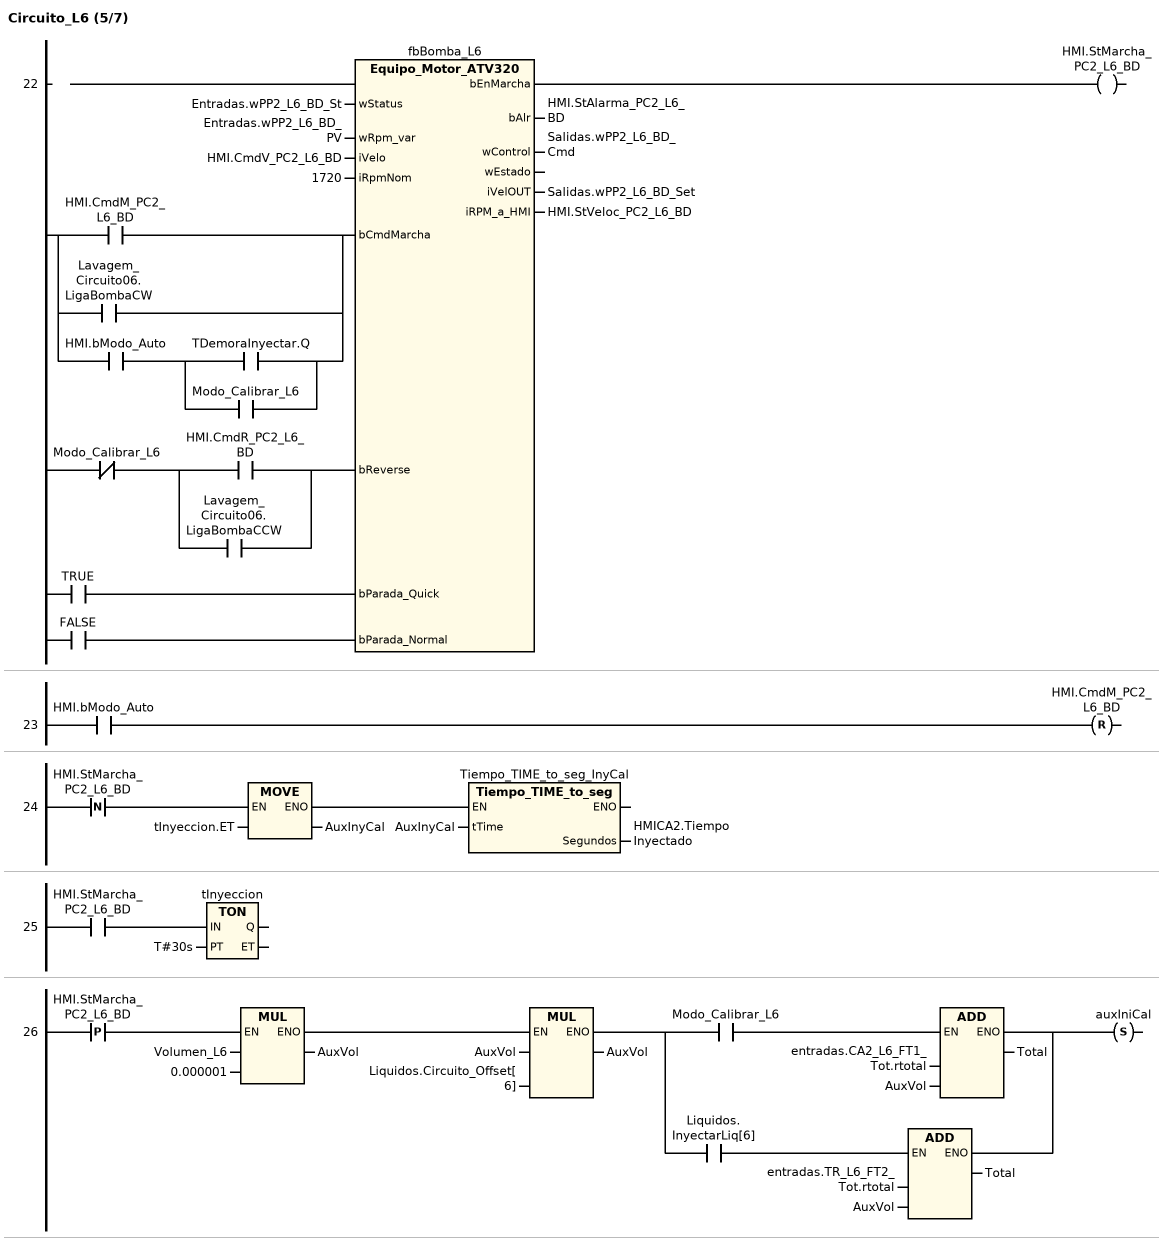
// NETWORK 22
fbBomba_L6(
    wStatus := Entradas.wPP2_L6_BD_St,
    wRpm_var := Entradas.wPP2_L6_BD_PV,
    iVelo := HMI.CmdV_PC2_L6_BD,
    iRpmNom := 1720,
    bCmdMarcha := HMI.CmdM_PC2_L6_BD OR Lavagem_Circuito06.LigaBombaCW OR HMI.bModo_Auto AND (TDemoraInyectar.Q OR Modo_Calibrar_L6),
    bReverse := NOT Modo_Calibrar_L6 AND (HMI.CmdR_PC2_L6_BD OR Lavagem_Circuito06.LigaBombaCCW),
    bParada_Quick := TRUE,
    bParada_Normal := FALSE,
    bAlr => HMI.StAlarma_PC2_L6_BD,
    wControl => Salidas.wPP2_L6_BD_Cmd,
    iVelOUT => Salidas.wPP2_L6_BD_Set,
    iRPM_a_HMI => HMI.StVeloc_PC2_L6_BD); // Equipo_Motor_ATV320
HMI.StMarcha_PC2_L6_BD := fbBomba_L6.bEnMarcha;

// NETWORK 23
HMI.CmdM_PC2_L6_BD R= HMI.bModo_Auto;

// NETWORK 24
_ft1(CLK := HMI.StMarcha_PC2_L6_BD);
_w8 := _ft1.Q;
IF _w8 THEN AuxInyCal := tInyeccion.ET; END_IF
IF _w8 THEN
    Tiempo_TIME_to_seg_InyCal(tTime := AuxInyCal, Segundos => HMICA2.TiempoInyectado); // Tiempo_TIME_to_seg
END_IF

// NETWORK 25
tInyeccion(IN := HMI.StMarcha_PC2_L6_BD, PT := T#30s); // TON

// NETWORK 26
_rt1(CLK := HMI.StMarcha_PC2_L6_BD);
_w9 := _rt1.Q;
IF _w9 THEN AuxVol := Volumen_L6 * 0.000001; END_IF
IF _w9 THEN AuxVol := AuxVol * Liquidos.Circuito_Offset[6]; END_IF
IF _w9 AND Modo_Calibrar_L6 THEN Total := entradas.CA2_L6_FT1_Tot.rtotal + AuxVol; END_IF
IF _w9 AND Liquidos.InyectarLiq[6] THEN Total := entradas.TR_L6_FT2_Tot.rtotal + AuxVol; END_IF
auxIniCal S= _w9 AND Modo_Calibrar_L6 OR _w9 AND Liquidos.InyectarLiq[6];

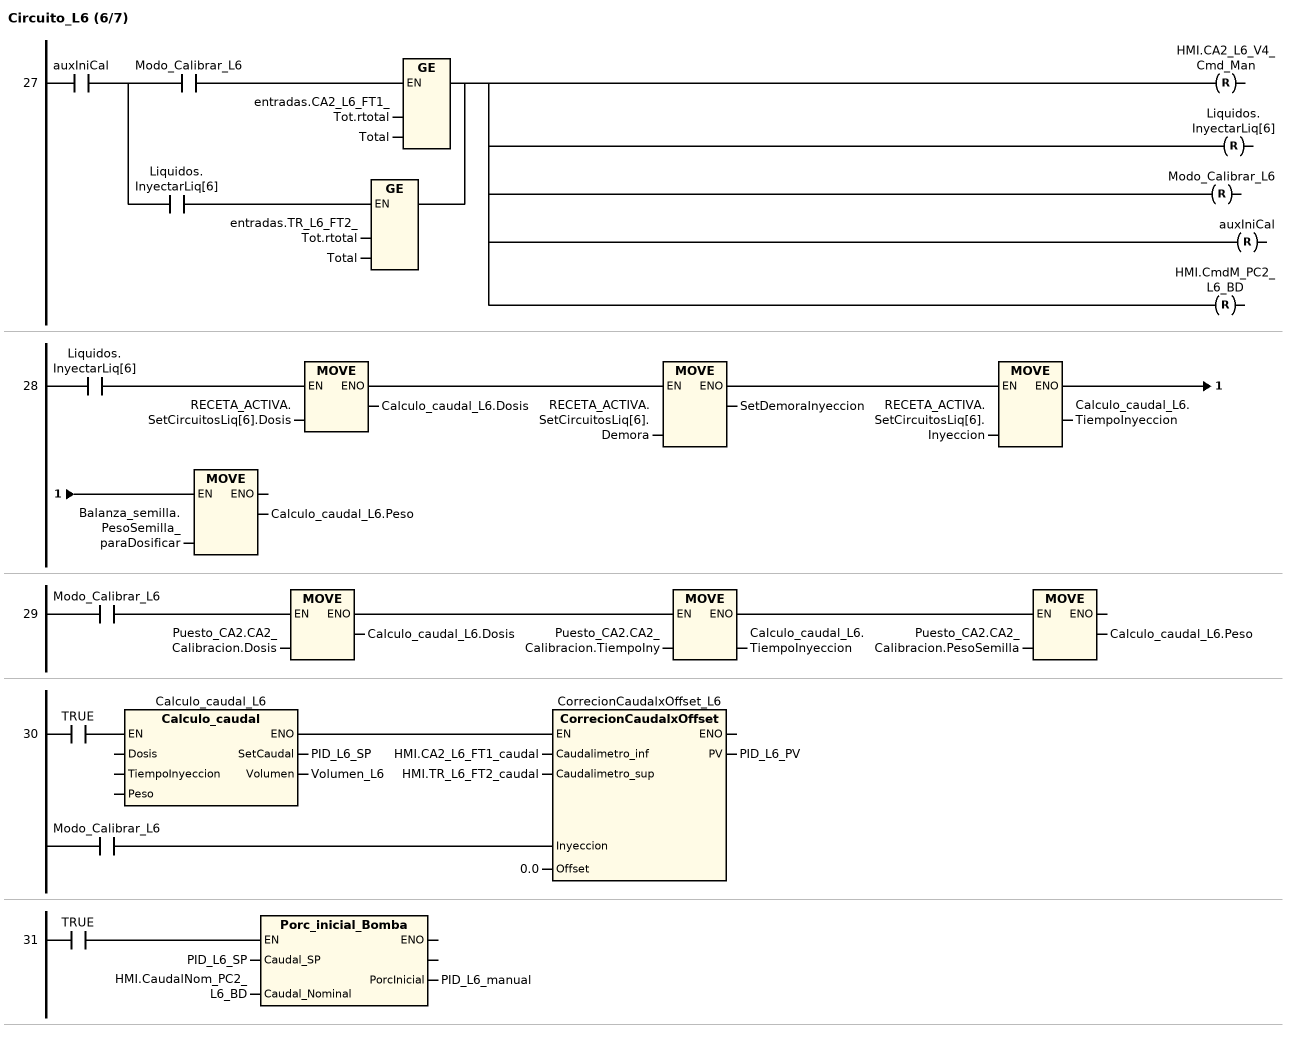
// NETWORK 27
_w10 := auxIniCal AND Modo_Calibrar_L6 AND entradas.CA2_L6_FT1_Tot.rtotal >= Total OR auxIniCal AND Liquidos.InyectarLiq[6] AND entradas.TR_L6_FT2_Tot.rtotal >= Total;
HMI.CA2_L6_V4_Cmd_Man R= _w10;
Liquidos.InyectarLiq[6] R= _w10;
Modo_Calibrar_L6 R= _w10;
auxIniCal R= _w10;
HMI.CmdM_PC2_L6_BD R= _w10;

// NETWORK 28
_w11 := Liquidos.InyectarLiq[6];
IF _w11 THEN Calculo_caudal_L6.Dosis := RECETA_ACTIVA.SetCircuitosLiq[6].Dosis; END_IF
IF _w11 THEN SetDemoraInyeccion := RECETA_ACTIVA.SetCircuitosLiq[6].Demora; END_IF
IF _w11 THEN Calculo_caudal_L6.TiempoInyeccion := RECETA_ACTIVA.SetCircuitosLiq[6].Inyeccion; END_IF
IF _w11 THEN Calculo_caudal_L6.Peso := Balanza_semilla.PesoSemilla_paraDosificar; END_IF

// NETWORK 29
_w12 := Modo_Calibrar_L6;
IF _w12 THEN Calculo_caudal_L6.Dosis := Puesto_CA2.CA2_Calibracion.Dosis; END_IF
IF _w12 THEN Calculo_caudal_L6.TiempoInyeccion := Puesto_CA2.CA2_Calibracion.TiempoIny; END_IF
IF _w12 THEN Calculo_caudal_L6.Peso := Puesto_CA2.CA2_Calibracion.PesoSemilla; END_IF

// NETWORK 30
Calculo_caudal_L6(SetCaudal => PID_L6_SP, Volumen => Volumen_L6); // Calculo_caudal
CorrecionCaudalxOffset_L6(
    Caudalimetro_inf := HMI.CA2_L6_FT1_caudal,
    Caudalimetro_sup := HMI.TR_L6_FT2_caudal,
    Inyeccion := Modo_Calibrar_L6,
    Offset := 0.0,
    PV => PID_L6_PV); // CorrecionCaudalxOffset

// NETWORK 31
Porc_inicial_Bomba(Caudal_SP := PID_L6_SP, Caudal_Nominal := HMI.CaudalNom_PC2_L6_BD, PorcInicial => PID_L6_manual);

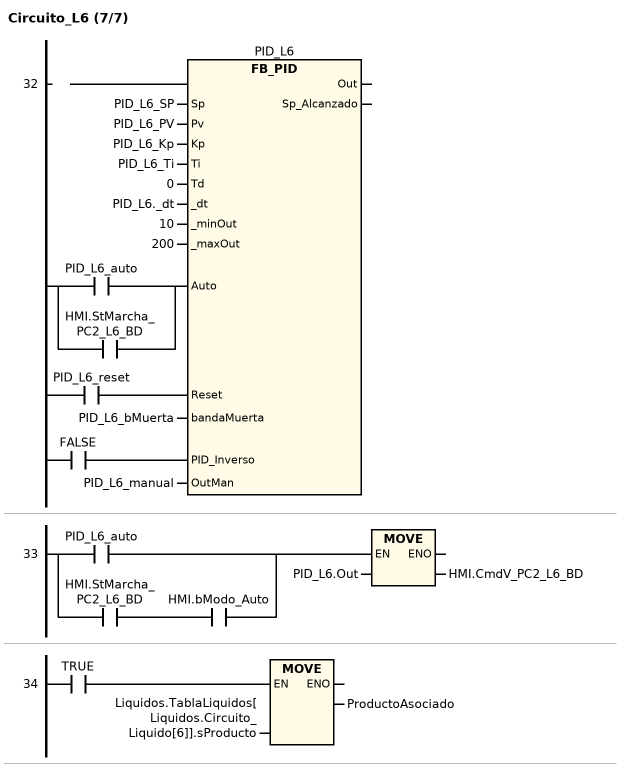
// NETWORK 32
PID_L6(
    Sp := PID_L6_SP,
    Pv := PID_L6_PV,
    Kp := PID_L6_Kp,
    Ti := PID_L6_Ti,
    Td := 0,
    _dt := PID_L6._dt,
    _minOut := 10,
    _maxOut := 200,
    Auto := PID_L6_auto OR HMI.StMarcha_PC2_L6_BD,
    Reset := PID_L6_reset,
    bandaMuerta := PID_L6_bMuerta,
    PID_Inverso := FALSE,
    OutMan := PID_L6_manual); // FB_PID

// NETWORK 33
IF PID_L6_auto OR HMI.StMarcha_PC2_L6_BD AND HMI.bModo_Auto THEN HMI.CmdV_PC2_L6_BD := PID_L6.Out; END_IF

// NETWORK 34
ProductoAsociado := Liquidos.TablaLiquidos[Liquidos.Circuito_Liquido[6]].sProducto;

END_PROGRAM

// ---- POUs/Puesto_Calibracion_2/Circuito_L7.TcPOU
PROGRAM Circuito_L7
VAR_INPUT
	Modo_Calibrar_L7: BOOL;
END_VAR
VAR
		fbBomba_L7 :Equipo_Motor_ATV320;
		ControlValv_ioLink_V1:ControlValv_ioLink;
		ControlValv_ioLink_V2: ControlValv_ioLink;
		ControlValv_ioLink_V3: ControlValv_ioLink;
		ControlValv_ioLink_V4: ControlValv_ioLink;
		Falla_L7_V1:BOOL;
		Falla_L7_V2:BOOL;
		Falla_L7_V3:BOOL;
		Falla_L7_V4:BOOL;
	Balanza_PU2_WT7: Balanza;
		dHS:DINT;
		TOF_calibradoIBC: TOF;
		PID_L7_SP:REAL;
		PID_L7_auto:BOOL;
		PID_L7_reset:BOOL;
		PID_L7_manual:REAL;
		PID_L7_bMuerta:REAL := 5;
		PID_L7_Kp:REAL := 0.1;
		PID_L7_Ti:REAL := 100;
		PID_L7_PV:REAL;
		Dosis_L7	:REAL;
		TiempoInyeccion_L7	:DINT;
		Peso	:REAL;
		Offset_L7:REAL;
		Inyeccion_L7:BOOL;
		Volumen_L7:REAL;
		Calculo_caudal_L7: Calculo_caudal;
		CorrecionCaudalxOffset_L7: CorrecionCaudalxOffset;
		tInyeccion: TON;
		Total :REAL;
		Totalant	:REAL;
		auxIniCal:BOOL;
		AuxVol:REAL;
		CA2_L7_V1_CmdA_Man :BOOL;
		CA2_L7_V4_CmdA_Man :BOOL;
		TDemoraInyectar: TON;
		SetDemoraInyeccion: REAL;
		Tiempo_seg_to_TIME_DemoraInyec: Tiempo_seg_to_TIME;
		AuxTDemoraInyec: TIME;
		PID_L7: FB_PID;
		Tiempo_TIME_to_seg_InyCal: Tiempo_TIME_to_seg;
		AuxInyCal:TIME;		
		IniTotalFT2:REAL;
		Auxconsumo:REAL;	
	ProductoAsociado: STRING;
	Lavagem_Circuito07: Lavagem;
	Calibracao_teste: Calibracao_V03;
END_VAR

VAR PERSISTENT
	UltimaCalibracao	:UDINT;	//Data e hora da ultima calibração
END_VAR
VAR // added by the converter: edge detectors and wires of the graphical bodies
    _w1, _w2, _w3, _w4, _w5, _w6, _w7, _w8, _w9, _w10, _w11, _w12, _w13 : BOOL;
    _ft1 : F_TRIG;
    _rt1, _rt2 : R_TRIG;
END_VAR

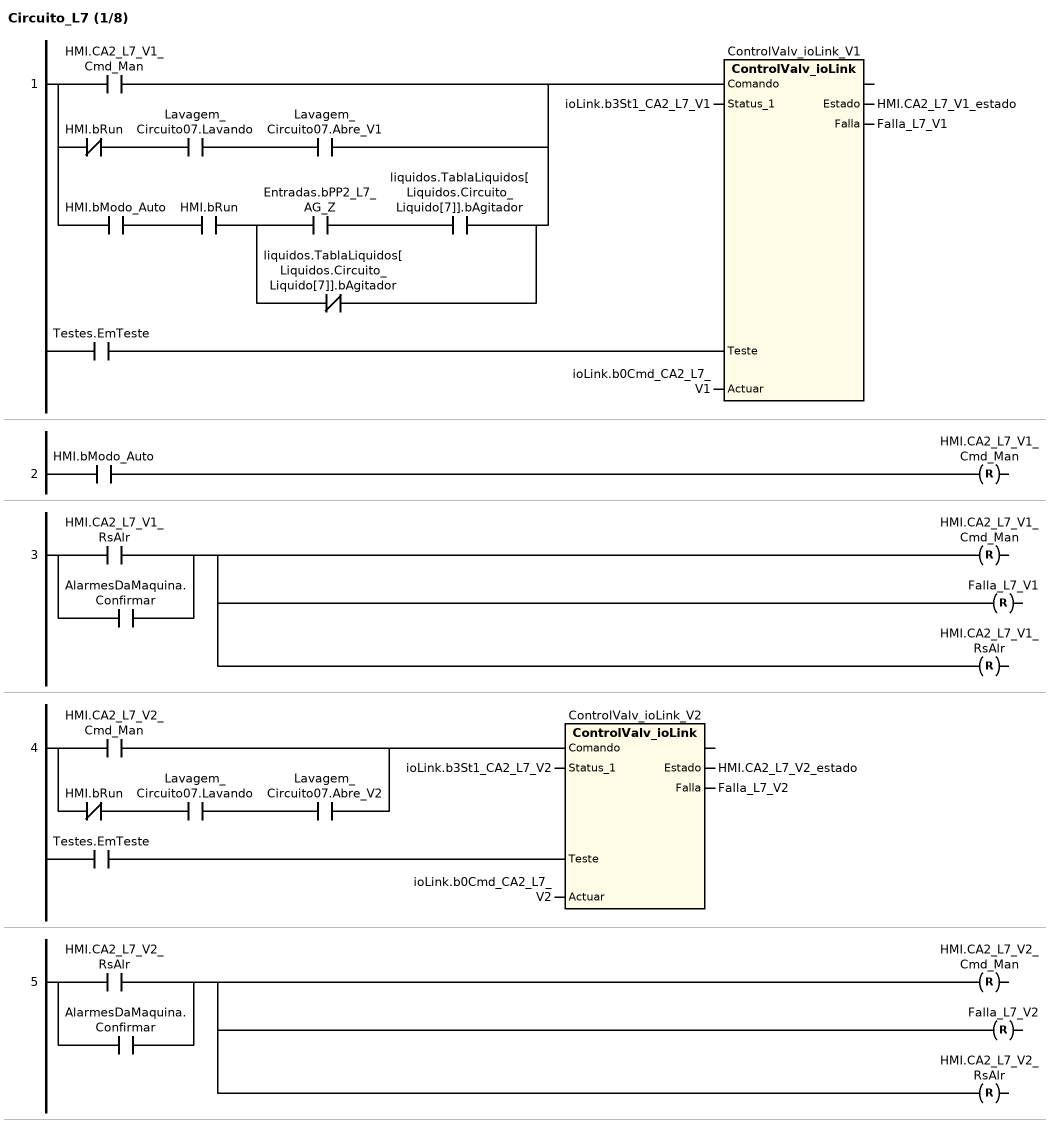
// NETWORK 1
ControlValv_ioLink_V1(
    Comando := HMI.CA2_L7_V1_Cmd_Man OR NOT HMI.bRun AND Lavagem_Circuito07.Lavando AND Lavagem_Circuito07.Abre_V1 OR HMI.bModo_Auto AND HMI.bRun AND (Entradas.bPP2_L7_AG_Z AND (liquidos.TablaLiquidos[Liquidos.Circuito_Liquido[7]].bAgitador) OR NOT (liquidos.TablaLiquidos[Liquidos.Circuito_Liquido[7]].bAgitador)),
    Status_1 := ioLink.b3St1_CA2_L7_V1,
    Teste := Testes.EmTeste,
    Actuar := ioLink.b0Cmd_CA2_L7_V1,
    Estado => HMI.CA2_L7_V1_estado,
    Falla => Falla_L7_V1); // ControlValv_ioLink

// NETWORK 2
HMI.CA2_L7_V1_Cmd_Man R= HMI.bModo_Auto;

// NETWORK 3
_w1 := HMI.CA2_L7_V1_RsAlr OR AlarmesDaMaquina.Confirmar;
HMI.CA2_L7_V1_Cmd_Man R= _w1;
Falla_L7_V1 R= _w1;
HMI.CA2_L7_V1_RsAlr R= _w1;

// NETWORK 4
ControlValv_ioLink_V2(
    Comando := HMI.CA2_L7_V2_Cmd_Man OR NOT HMI.bRun AND Lavagem_Circuito07.Lavando AND Lavagem_Circuito07.Abre_V2,
    Status_1 := ioLink.b3St1_CA2_L7_V2,
    Teste := Testes.EmTeste,
    Actuar := ioLink.b0Cmd_CA2_L7_V2,
    Estado => HMI.CA2_L7_V2_estado,
    Falla => Falla_L7_V2); // ControlValv_ioLink

// NETWORK 5
_w2 := HMI.CA2_L7_V2_RsAlr OR AlarmesDaMaquina.Confirmar;
HMI.CA2_L7_V2_Cmd_Man R= _w2;
Falla_L7_V2 R= _w2;
HMI.CA2_L7_V2_RsAlr R= _w2;

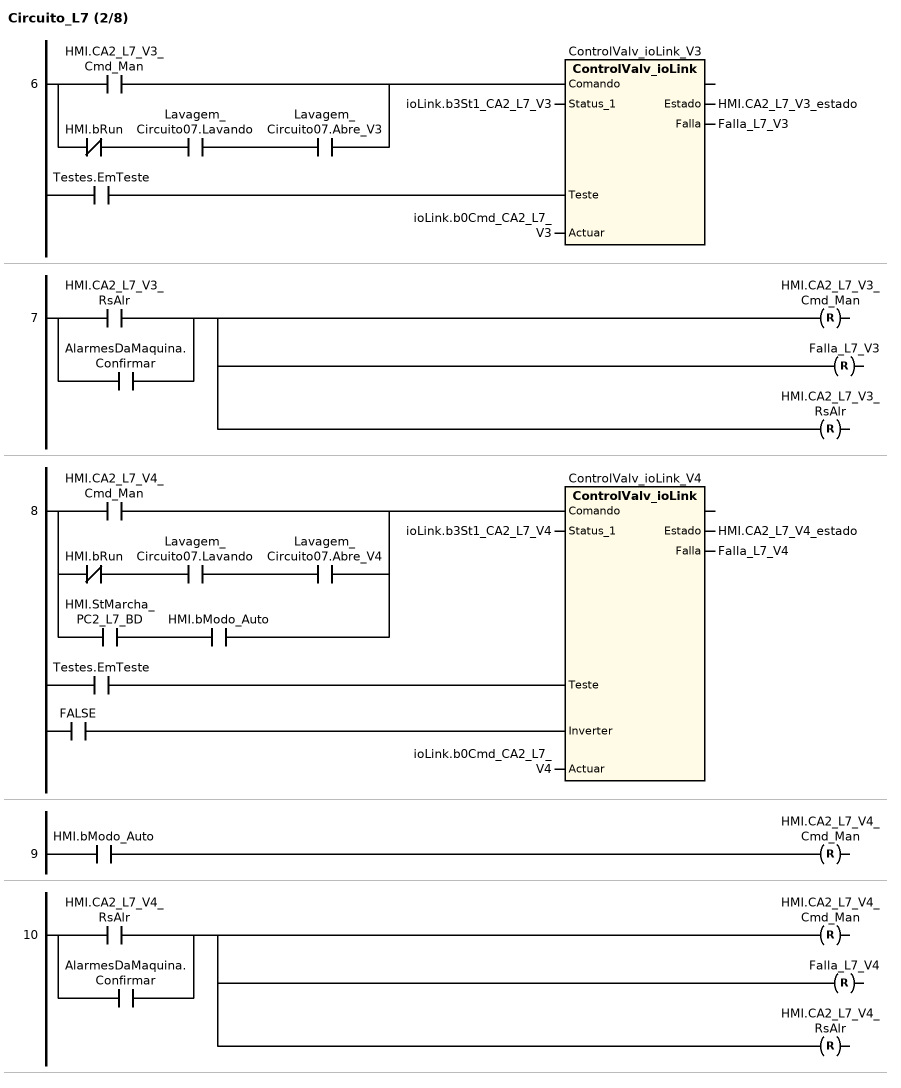
// NETWORK 6
ControlValv_ioLink_V3(
    Comando := HMI.CA2_L7_V3_Cmd_Man OR NOT HMI.bRun AND Lavagem_Circuito07.Lavando AND Lavagem_Circuito07.Abre_V3,
    Status_1 := ioLink.b3St1_CA2_L7_V3,
    Teste := Testes.EmTeste,
    Actuar := ioLink.b0Cmd_CA2_L7_V3,
    Estado => HMI.CA2_L7_V3_estado,
    Falla => Falla_L7_V3); // ControlValv_ioLink

// NETWORK 7
_w3 := HMI.CA2_L7_V3_RsAlr OR AlarmesDaMaquina.Confirmar;
HMI.CA2_L7_V3_Cmd_Man R= _w3;
Falla_L7_V3 R= _w3;
HMI.CA2_L7_V3_RsAlr R= _w3;

// NETWORK 8
ControlValv_ioLink_V4(
    Comando := HMI.CA2_L7_V4_Cmd_Man OR NOT HMI.bRun AND Lavagem_Circuito07.Lavando AND Lavagem_Circuito07.Abre_V4 OR HMI.StMarcha_PC2_L7_BD AND HMI.bModo_Auto,
    Status_1 := ioLink.b3St1_CA2_L7_V4,
    Teste := Testes.EmTeste,
    Inverter := FALSE,
    Actuar := ioLink.b0Cmd_CA2_L7_V4,
    Estado => HMI.CA2_L7_V4_estado,
    Falla => Falla_L7_V4); // ControlValv_ioLink

// NETWORK 9
HMI.CA2_L7_V4_Cmd_Man R= HMI.bModo_Auto;

// NETWORK 10
_w4 := HMI.CA2_L7_V4_RsAlr OR AlarmesDaMaquina.Confirmar;
HMI.CA2_L7_V4_Cmd_Man R= _w4;
Falla_L7_V4 R= _w4;
HMI.CA2_L7_V4_RsAlr R= _w4;

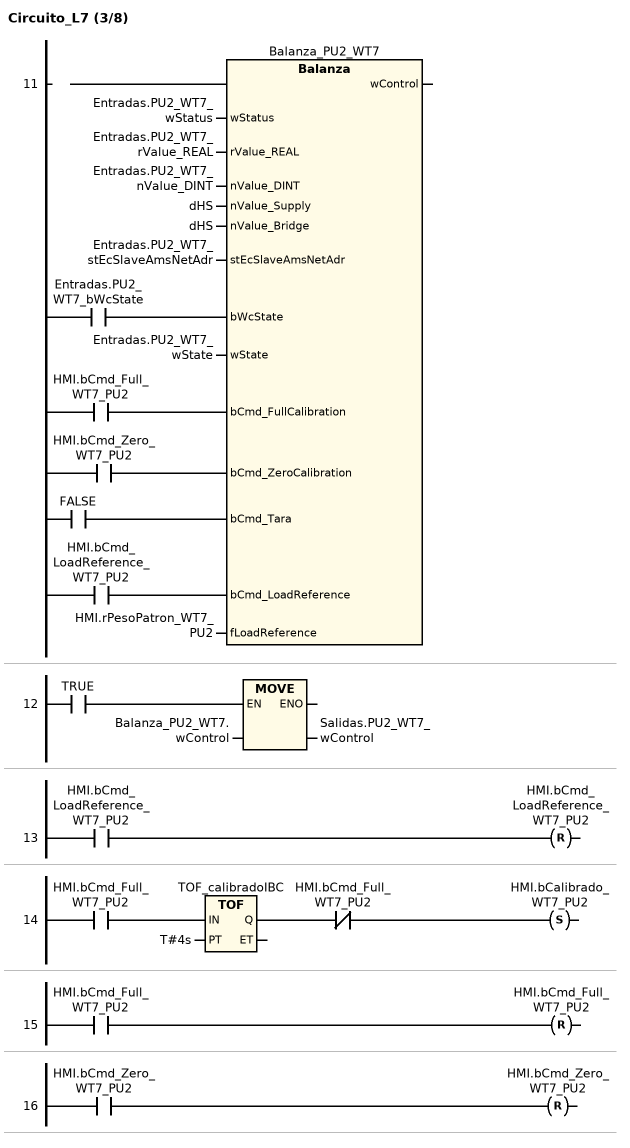
// NETWORK 11
Balanza_PU2_WT7(
    wStatus := Entradas.PU2_WT7_wStatus,
    rValue_REAL := Entradas.PU2_WT7_rValue_REAL,
    nValue_DINT := Entradas.PU2_WT7_nValue_DINT,
    nValue_Supply := dHS,
    nValue_Bridge := dHS,
    stEcSlaveAmsNetAdr := Entradas.PU2_WT7_stEcSlaveAmsNetAdr,
    bWcState := Entradas.PU2_WT7_bWcState,
    wState := Entradas.PU2_WT7_wState,
    bCmd_FullCalibration := HMI.bCmd_Full_WT7_PU2,
    bCmd_ZeroCalibration := HMI.bCmd_Zero_WT7_PU2,
    bCmd_Tara := FALSE,
    bCmd_LoadReference := HMI.bCmd_LoadReference_WT7_PU2,
    fLoadReference := HMI.rPesoPatron_WT7_PU2); // Balanza

// NETWORK 12
Salidas.PU2_WT7_wControl := Balanza_PU2_WT7.wControl;

// NETWORK 13
HMI.bCmd_LoadReference_WT7_PU2 R= HMI.bCmd_LoadReference_WT7_PU2;

// NETWORK 14
TOF_calibradoIBC(IN := HMI.bCmd_Full_WT7_PU2, PT := T#4s); // TOF
HMI.bCalibrado_WT7_PU2 S= TOF_calibradoIBC.Q AND NOT HMI.bCmd_Full_WT7_PU2;

// NETWORK 15
HMI.bCmd_Full_WT7_PU2 R= HMI.bCmd_Full_WT7_PU2;

// NETWORK 16
HMI.bCmd_Zero_WT7_PU2 R= HMI.bCmd_Zero_WT7_PU2;

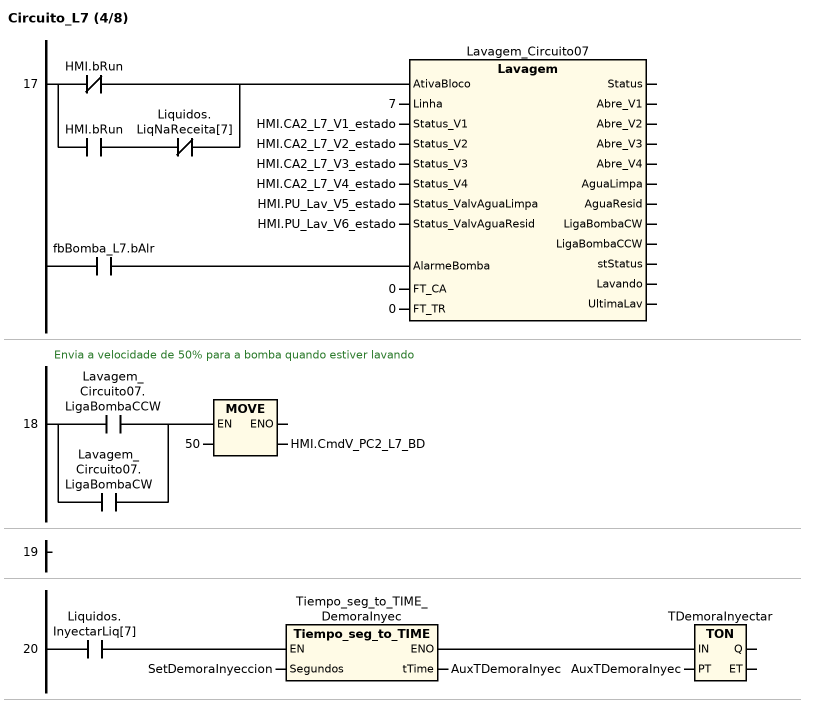
// NETWORK 17
Lavagem_Circuito07(
    AtivaBloco := NOT HMI.bRun OR HMI.bRun AND NOT Liquidos.LiqNaReceita[7],
    Linha := 7,
    Status_V1 := HMI.CA2_L7_V1_estado,
    Status_V2 := HMI.CA2_L7_V2_estado,
    Status_V3 := HMI.CA2_L7_V3_estado,
    Status_V4 := HMI.CA2_L7_V4_estado,
    Status_ValvAguaLimpa := HMI.PU_Lav_V5_estado,
    Status_ValvAguaResid := HMI.PU_Lav_V6_estado,
    AlarmeBomba := fbBomba_L7.bAlr,
    FT_CA := 0,
    FT_TR := 0); // Lavagem

// NETWORK 18
// Envia a velocidade de 50% para a bomba quando estiver lavando
IF Lavagem_Circuito07.LigaBombaCCW OR Lavagem_Circuito07.LigaBombaCW THEN HMI.CmdV_PC2_L7_BD := 50; END_IF

// NETWORK 19

// NETWORK 20
_w5 := Liquidos.InyectarLiq[7];
IF _w5 THEN
    Tiempo_seg_to_TIME_DemoraInyec(Segundos := SetDemoraInyeccion, tTime => AuxTDemoraInyec); // Tiempo_seg_to_TIME
END_IF
TDemoraInyectar(IN := _w5, PT := AuxTDemoraInyec); // TON

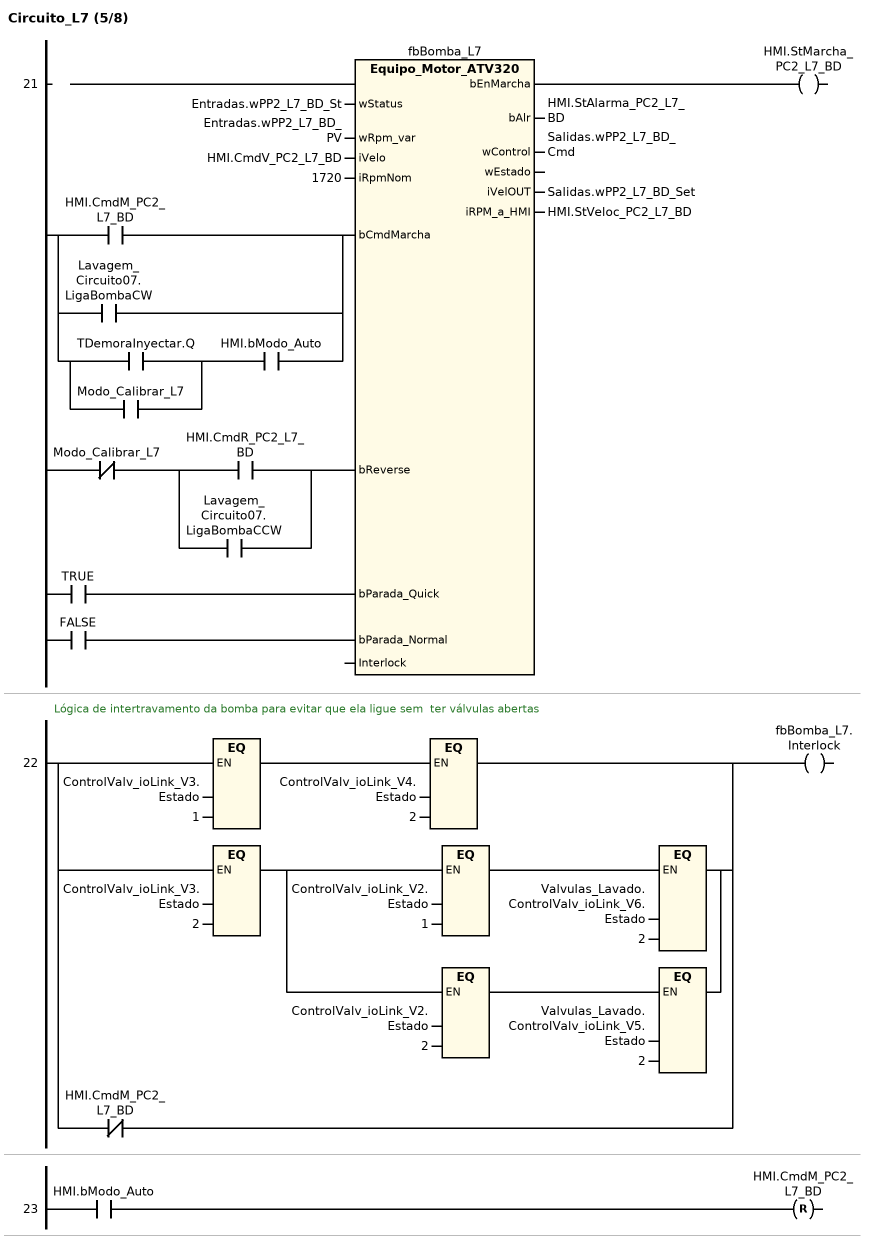
// NETWORK 21
fbBomba_L7(
    wStatus := Entradas.wPP2_L7_BD_St,
    wRpm_var := Entradas.wPP2_L7_BD_PV,
    iVelo := HMI.CmdV_PC2_L7_BD,
    iRpmNom := 1720,
    bCmdMarcha := HMI.CmdM_PC2_L7_BD OR Lavagem_Circuito07.LigaBombaCW OR (TDemoraInyectar.Q OR Modo_Calibrar_L7) AND HMI.bModo_Auto,
    bReverse := NOT Modo_Calibrar_L7 AND (HMI.CmdR_PC2_L7_BD OR Lavagem_Circuito07.LigaBombaCCW),
    bParada_Quick := TRUE,
    bParada_Normal := FALSE,
    bAlr => HMI.StAlarma_PC2_L7_BD,
    wControl => Salidas.wPP2_L7_BD_Cmd,
    iVelOUT => Salidas.wPP2_L7_BD_Set,
    iRPM_a_HMI => HMI.StVeloc_PC2_L7_BD); // Equipo_Motor_ATV320
HMI.StMarcha_PC2_L7_BD := fbBomba_L7.bEnMarcha;

// NETWORK 22
// Lógica de intertravamento da bomba para evitar que ela ligue sem  ter válvulas abertas
_w6 := NOT HMI.CmdM_PC2_L7_BD;
IF NOT _w6 THEN
    _w7 := ControlValv_ioLink_V3.Estado = 2;
    _w6 := ControlValv_ioLink_V3.Estado = 1 AND ControlValv_ioLink_V4.Estado = 2 OR (_w7 AND ControlValv_ioLink_V2.Estado = 1 AND Valvulas_Lavado.ControlValv_ioLink_V6.Estado = 2 OR _w7 AND ControlValv_ioLink_V2.Estado = 2 AND Valvulas_Lavado.ControlValv_ioLink_V5.Estado = 2);
END_IF
fbBomba_L7.Interlock := _w6;

// NETWORK 23
HMI.CmdM_PC2_L7_BD R= HMI.bModo_Auto;

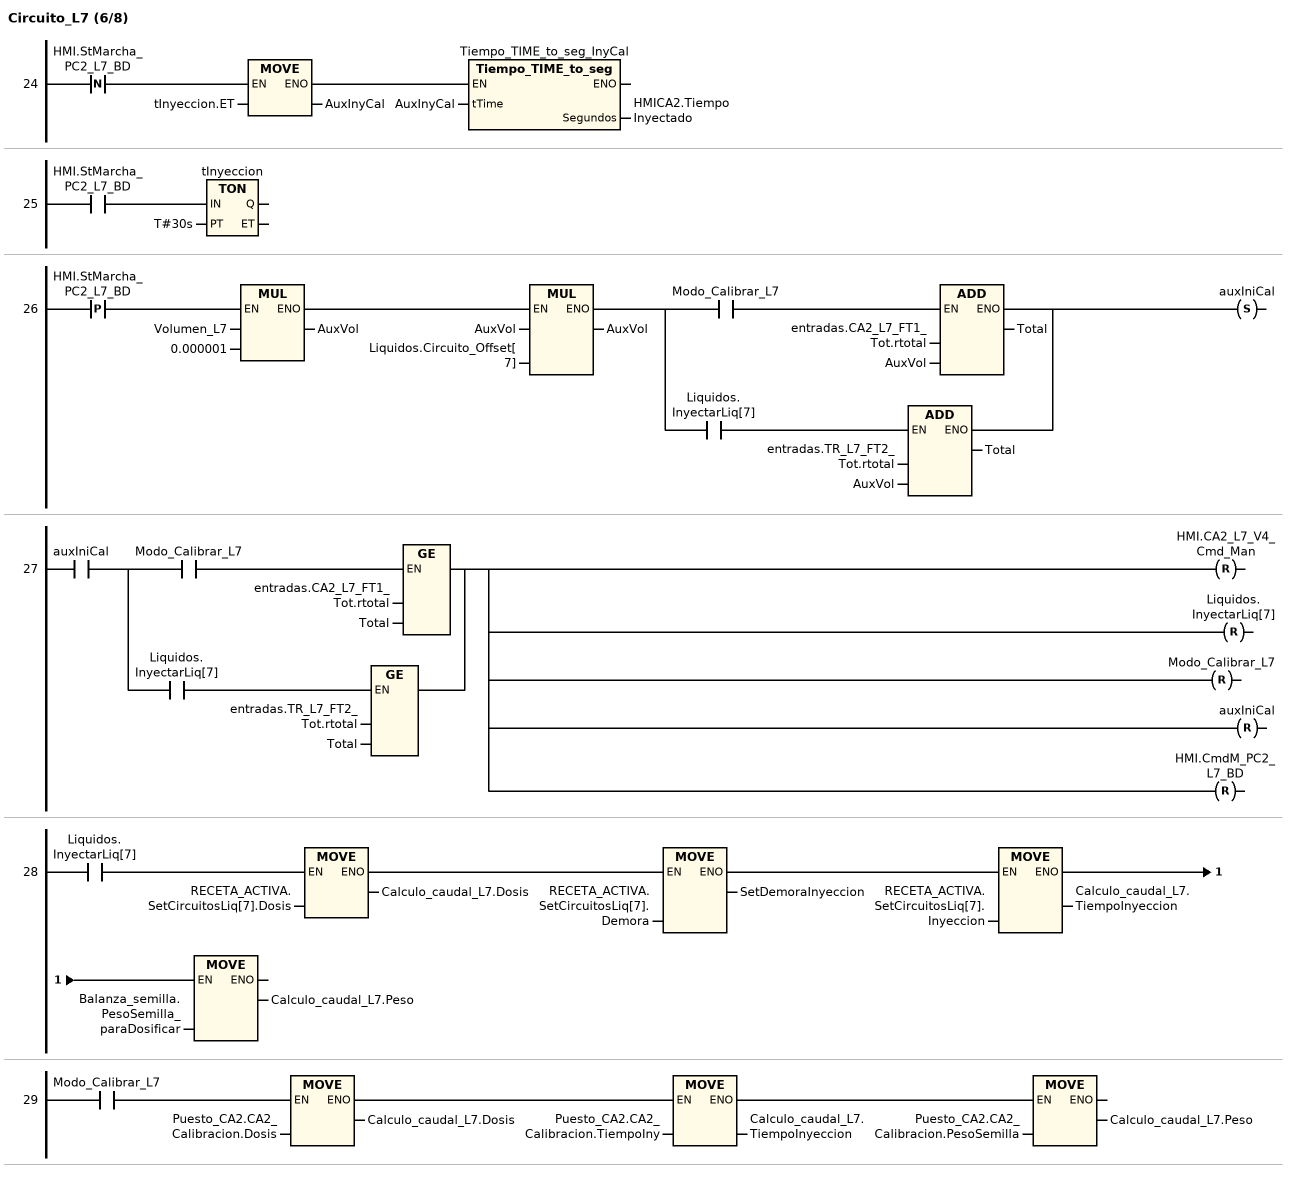
// NETWORK 24
_ft1(CLK := HMI.StMarcha_PC2_L7_BD);
_w8 := _ft1.Q;
IF _w8 THEN AuxInyCal := tInyeccion.ET; END_IF
IF _w8 THEN
    Tiempo_TIME_to_seg_InyCal(tTime := AuxInyCal, Segundos => HMICA2.TiempoInyectado); // Tiempo_TIME_to_seg
END_IF

// NETWORK 25
tInyeccion(IN := HMI.StMarcha_PC2_L7_BD, PT := T#30s); // TON

// NETWORK 26
_rt1(CLK := HMI.StMarcha_PC2_L7_BD);
_w9 := _rt1.Q;
IF _w9 THEN AuxVol := Volumen_L7 * 0.000001; END_IF
IF _w9 THEN AuxVol := AuxVol * Liquidos.Circuito_Offset[7]; END_IF
IF _w9 AND Modo_Calibrar_L7 THEN Total := entradas.CA2_L7_FT1_Tot.rtotal + AuxVol; END_IF
IF _w9 AND Liquidos.InyectarLiq[7] THEN Total := entradas.TR_L7_FT2_Tot.rtotal + AuxVol; END_IF
auxIniCal S= _w9 AND Modo_Calibrar_L7 OR _w9 AND Liquidos.InyectarLiq[7];

// NETWORK 27
_w10 := auxIniCal AND Modo_Calibrar_L7 AND entradas.CA2_L7_FT1_Tot.rtotal >= Total OR auxIniCal AND Liquidos.InyectarLiq[7] AND entradas.TR_L7_FT2_Tot.rtotal >= Total;
HMI.CA2_L7_V4_Cmd_Man R= _w10;
Liquidos.InyectarLiq[7] R= _w10;
Modo_Calibrar_L7 R= _w10;
auxIniCal R= _w10;
HMI.CmdM_PC2_L7_BD R= _w10;

// NETWORK 28
_w11 := Liquidos.InyectarLiq[7];
IF _w11 THEN Calculo_caudal_L7.Dosis := RECETA_ACTIVA.SetCircuitosLiq[7].Dosis; END_IF
IF _w11 THEN SetDemoraInyeccion := RECETA_ACTIVA.SetCircuitosLiq[7].Demora; END_IF
IF _w11 THEN Calculo_caudal_L7.TiempoInyeccion := RECETA_ACTIVA.SetCircuitosLiq[7].Inyeccion; END_IF
IF _w11 THEN Calculo_caudal_L7.Peso := Balanza_semilla.PesoSemilla_paraDosificar; END_IF

// NETWORK 29
_w12 := Modo_Calibrar_L7;
IF _w12 THEN Calculo_caudal_L7.Dosis := Puesto_CA2.CA2_Calibracion.Dosis; END_IF
IF _w12 THEN Calculo_caudal_L7.TiempoInyeccion := Puesto_CA2.CA2_Calibracion.TiempoIny; END_IF
IF _w12 THEN Calculo_caudal_L7.Peso := Puesto_CA2.CA2_Calibracion.PesoSemilla; END_IF

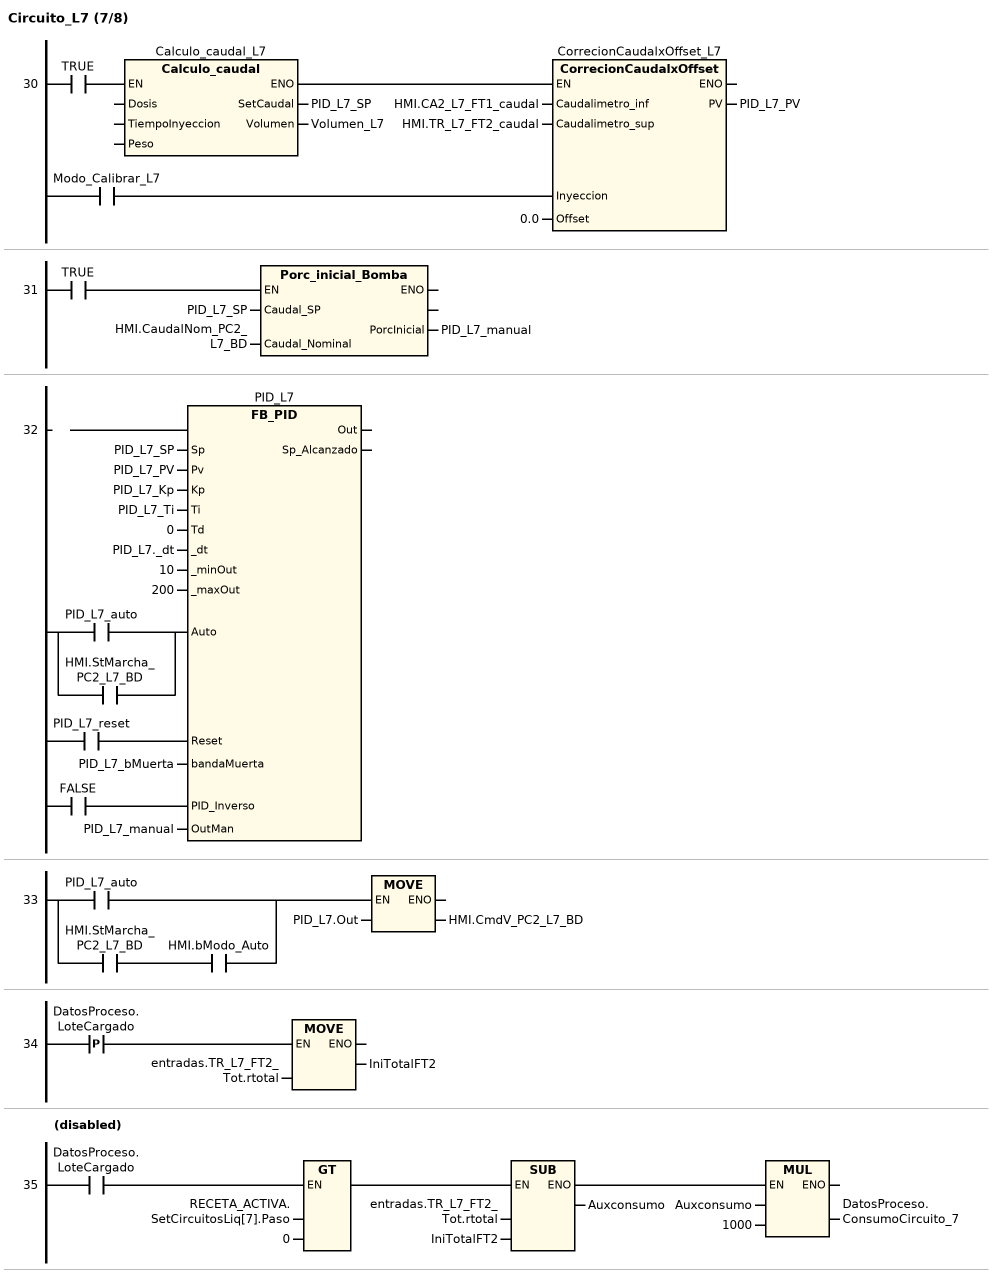
// NETWORK 30
Calculo_caudal_L7(SetCaudal => PID_L7_SP, Volumen => Volumen_L7); // Calculo_caudal
CorrecionCaudalxOffset_L7(
    Caudalimetro_inf := HMI.CA2_L7_FT1_caudal,
    Caudalimetro_sup := HMI.TR_L7_FT2_caudal,
    Inyeccion := Modo_Calibrar_L7,
    Offset := 0.0,
    PV => PID_L7_PV); // CorrecionCaudalxOffset

// NETWORK 31
Porc_inicial_Bomba(Caudal_SP := PID_L7_SP, Caudal_Nominal := HMI.CaudalNom_PC2_L7_BD, PorcInicial => PID_L7_manual);

// NETWORK 32
PID_L7(
    Sp := PID_L7_SP,
    Pv := PID_L7_PV,
    Kp := PID_L7_Kp,
    Ti := PID_L7_Ti,
    Td := 0,
    _dt := PID_L7._dt,
    _minOut := 10,
    _maxOut := 200,
    Auto := PID_L7_auto OR HMI.StMarcha_PC2_L7_BD,
    Reset := PID_L7_reset,
    bandaMuerta := PID_L7_bMuerta,
    PID_Inverso := FALSE,
    OutMan := PID_L7_manual); // FB_PID

// NETWORK 33
IF PID_L7_auto OR HMI.StMarcha_PC2_L7_BD AND HMI.bModo_Auto THEN HMI.CmdV_PC2_L7_BD := PID_L7.Out; END_IF

// NETWORK 34
_rt2(CLK := DatosProceso.LoteCargado);
IF _rt2.Q THEN IniTotalFT2 := entradas.TR_L7_FT2_Tot.rtotal; END_IF

// NETWORK 35 (disabled)
// _w13 := DatosProceso.LoteCargado AND RECETA_ACTIVA.SetCircuitosLiq[7].Paso > 0;
// IF _w13 THEN Auxconsumo := entradas.TR_L7_FT2_Tot.rtotal - IniTotalFT2; END_IF
// IF _w13 THEN DatosProceso.ConsumoCircuito_7 := Auxconsumo * 1000; END_IF

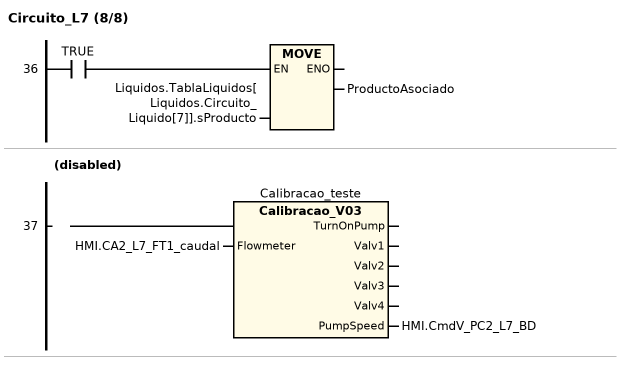
// NETWORK 36
ProductoAsociado := Liquidos.TablaLiquidos[Liquidos.Circuito_Liquido[7]].sProducto;

// NETWORK 37 (disabled)
// Calibracao_teste(Flowmeter := HMI.CA2_L7_FT1_caudal, PumpSpeed => HMI.CmdV_PC2_L7_BD); // Calibracao_V03

END_PROGRAM

// ---- POUs/Testes Thiago/Calibracao_V03.TcPOU
FUNCTION_BLOCK Calibracao_V03
VAR_INPUT
	Flowmeter:REAL;
END_VAR
VAR_OUTPUT
	TurnOnPump:BOOL;
	Valv1:BOOL;
	Valv2:BOOL;
	Valv3:BOOL;
	Valv4:BOOL;
	PumpSpeed:REAL;	//Velocidade enviada para a bomba
END_VAR
VAR
	SwitchCase:INT;
	Start: BOOL;
	Stop: BOOL;
	TON_Temporizador1: TON;
	TON_Temporizador2: TON;
	BaixaVazao	:ARRAY[1..10] OF REAL;
	AltaVazao	:ARRAY[1..10] OF REAL;
	MediaBaixaVazao :REAL;
	MediaAltaVazao	:REAL;
	Counter: INT;
	i: INT;
	CoefAngular: REAL;
END_VAR

//Esse programa encontrará dois pontos relacionando vazão e velocidade (x e y), assim, será possível definir a função da bomba

IF Start AND NOT Stop  AND Seguridad.PB_Emergencia THEN
	SwitchCase := 10;
	Start := FALSE;
END_IF

IF STOP OR NOT Seguridad.PB_Emergencia THEN
	SwitchCase := 0;
	STOP := FALSE;
END_IF

//Temporizadores
TON_Temporizador1(PT:=T#5S);
TON_Temporizador2( IN:=TON_Temporizador1.Q AND NOT TON_Temporizador2.Q, PT:=T#1S);


CASE SwitchCase OF
	0:	//Desliga o sistema
		TurnOnPump := FALSE;
		Valv1 := FALSE;
		Valv2 := FALSE;
		Valv3 := FALSE;
		Valv4 := FALSE;
		
	10:	//Inicia a bomba com 20%
		PumpSpeed := 20;
		TurnOnPump := TRUE;
		TON_Temporizador1.IN := TRUE;
		
		//Após 5s da bomba ligada, a vazão é computada a cada 1s
		IF TON_Temporizador1.Q THEN
			Counter := 1;
			SwitchCase := 20;
		END_IF
		
	20:	//Cômputo da vazão com 10% da velocidade e aguarda a estabilização
		IF TON_Temporizador2.Q THEN
			IF Flowmeter > 0 THEN
				BaixaVazao[Counter] := Flowmeter;
				Counter := Counter + 1;
			END_IF
		END_IF
		IF Counter > 10 THEN
			TON_Temporizador1.IN := FALSE;
			SwitchCase := 30;
		END_IF
	
	30:	//Inicia a bomba com 80% e aguarda a estabilização
		PumpSpeed := 80;
		TON_Temporizador1.IN := TRUE;
		IF TON_Temporizador1.Q THEN
			Counter := 1;
			SwitchCase := 40;
		END_IF
		
	40:	//Cômputo da vazão com 80% da velocidade
		IF TON_Temporizador2.Q THEN
			IF Flowmeter > 0 THEN
				AltaVazao[Counter] := Flowmeter;
				Counter := Counter + 1;
			END_IF
		END_IF
		IF Counter > 10 THEN
			TON_Temporizador1.IN := FALSE;
			SwitchCase := 50;
		END_IF
		
	50:	//Cálculo das médias
		MediaBaixaVazao	:= 0;
		MediaAltaVazao	:= 0;
		FOR i := 1 TO 10 BY 1 DO
			MediaBaixaVazao	:= MediaBaixaVazao + BaixaVazao[i];
			MediaAltaVazao	:= MediaAltaVazao + AltaVazao[i];
		END_FOR
		MediaBaixaVazao	:= MediaBaixaVazao/10;
		MediaAltaVazao	:= MediaAltaVazao/10;
		
		//Cálculo do coeficiente angular
		CoefAngular := (MediaAltaVazao - MediaBaixaVazao)/(80 - 20);
		TurnOnPump := FALSE;
		SwitchCase := 0;
		
	60:	//
		
END_CASE

END_FUNCTION_BLOCK

// ---- POUs/Puesto_Calibracion_2/Circuito_L8.TcPOU
PROGRAM Circuito_L8
VAR_INPUT
	Modo_Calibrar_L8: BOOL;
END_VAR
VAR
		fbBomba_L8 :Equipo_Motor_ATV320;
		ControlValv_ioLink_V1:ControlValv_ioLink;
		ControlValv_ioLink_V2: ControlValv_ioLink;
		ControlValv_ioLink_V3: ControlValv_ioLink;
		ControlValv_ioLink_V4: ControlValv_ioLink;
		Falla_L8_V1:BOOL;
		Falla_L8_V2:BOOL;
		Falla_L8_V3:BOOL;
		Falla_L8_V4:BOOL;
	Balanza_PU2_WT8: Balanza;
		dHS:DINT;
		TOF_calibradoIBC: TOF;
		PID_L8_SP:REAL;
		PID_L8_auto:BOOL;
		PID_L8_reset:BOOL;
		PID_L8_manual:REAL;
		PID_L8_bMuerta:REAL := 5;
		PID_L8_Kp:REAL := 0.1;
		PID_L8_Ti:REAL := 100;
		PID_L8_PV:REAL;
		Dosis_L8	:REAL;
		TiempoInyeccion_L8	:DINT;
		Peso	:REAL;
		Offset_L8:REAL;
		Inyeccion_L8:BOOL;
		Volumen_L8:REAL;
		Calculo_caudal_L8: Calculo_caudal;
		CorrecionCaudalxOffset_L8: CorrecionCaudalxOffset;
		tInyeccion: TON;
		Total :REAL;
		Totalant	:REAL;
		auxIniCal:BOOL;
		AuxVol:REAL;
		CA2_L8_V1_CmdA_Man :BOOL;
		CA2_L8_V4_CmdA_Man :BOOL;
		TDemoraInyectar: TON;
		SetDemoraInyeccion: REAL;
		Tiempo_seg_to_TIME_DemoraInyec: Tiempo_seg_to_TIME;
		AuxTDemoraInyec: TIME;
		PID_L8: FB_PID;		
		Tiempo_TIME_to_seg_InyCal: Tiempo_TIME_to_seg;
		AuxInyCal:TIME;	
		IniTotalFT2:REAL;
		Auxconsumo:REAL;
	ProductoAsociado: STRING;
	Lavagem_Circuito08: Lavagem;
	FB_BasicPID_0: FB_BasicPID;
	Teste: BOOL;
END_VAR

VAR PERSISTENT
	UltimaCalibracao	:UDINT;	//Data e hora da ultima calibração
END_VAR
VAR // added by the converter: edge detectors and wires of the graphical bodies
    _w1, _w2, _w3, _w4, _w5, _w6, _w7, _w8, _w9, _w10, _w11, _w12, _w13 : BOOL;
    _ft1 : F_TRIG;
    _rt1, _rt2 : R_TRIG;
END_VAR

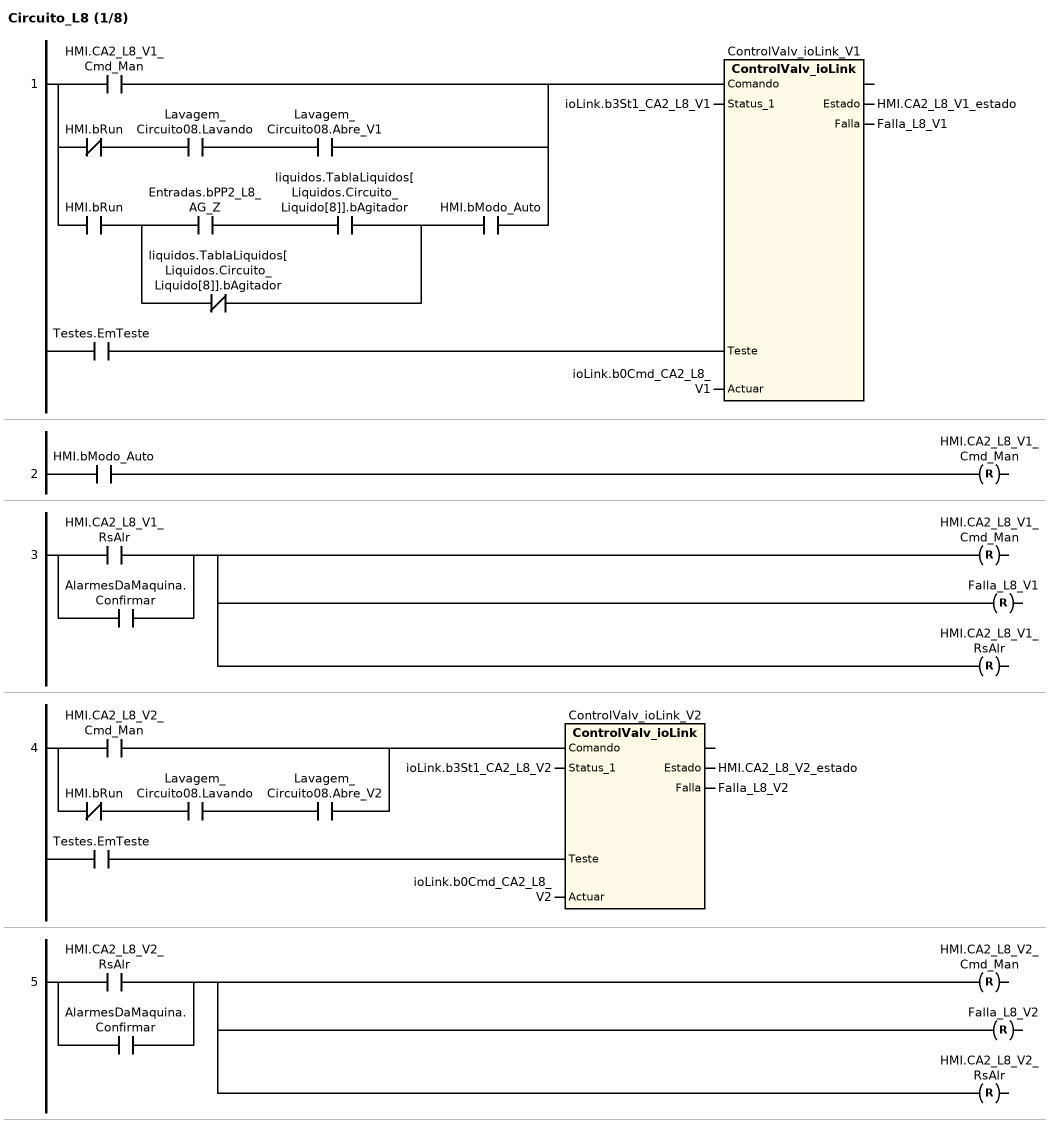
// NETWORK 1
ControlValv_ioLink_V1(
    Comando := HMI.CA2_L8_V1_Cmd_Man OR NOT HMI.bRun AND Lavagem_Circuito08.Lavando AND Lavagem_Circuito08.Abre_V1 OR HMI.bRun AND (Entradas.bPP2_L8_AG_Z AND (liquidos.TablaLiquidos[Liquidos.Circuito_Liquido[8]].bAgitador) OR NOT (liquidos.TablaLiquidos[Liquidos.Circuito_Liquido[8]].bAgitador)) AND HMI.bModo_Auto,
    Status_1 := ioLink.b3St1_CA2_L8_V1,
    Teste := Testes.EmTeste,
    Actuar := ioLink.b0Cmd_CA2_L8_V1,
    Estado => HMI.CA2_L8_V1_estado,
    Falla => Falla_L8_V1); // ControlValv_ioLink

// NETWORK 2
HMI.CA2_L8_V1_Cmd_Man R= HMI.bModo_Auto;

// NETWORK 3
_w1 := HMI.CA2_L8_V1_RsAlr OR AlarmesDaMaquina.Confirmar;
HMI.CA2_L8_V1_Cmd_Man R= _w1;
Falla_L8_V1 R= _w1;
HMI.CA2_L8_V1_RsAlr R= _w1;

// NETWORK 4
ControlValv_ioLink_V2(
    Comando := HMI.CA2_L8_V2_Cmd_Man OR NOT HMI.bRun AND Lavagem_Circuito08.Lavando AND Lavagem_Circuito08.Abre_V2,
    Status_1 := ioLink.b3St1_CA2_L8_V2,
    Teste := Testes.EmTeste,
    Actuar := ioLink.b0Cmd_CA2_L8_V2,
    Estado => HMI.CA2_L8_V2_estado,
    Falla => Falla_L8_V2); // ControlValv_ioLink

// NETWORK 5
_w2 := HMI.CA2_L8_V2_RsAlr OR AlarmesDaMaquina.Confirmar;
HMI.CA2_L8_V2_Cmd_Man R= _w2;
Falla_L8_V2 R= _w2;
HMI.CA2_L8_V2_RsAlr R= _w2;

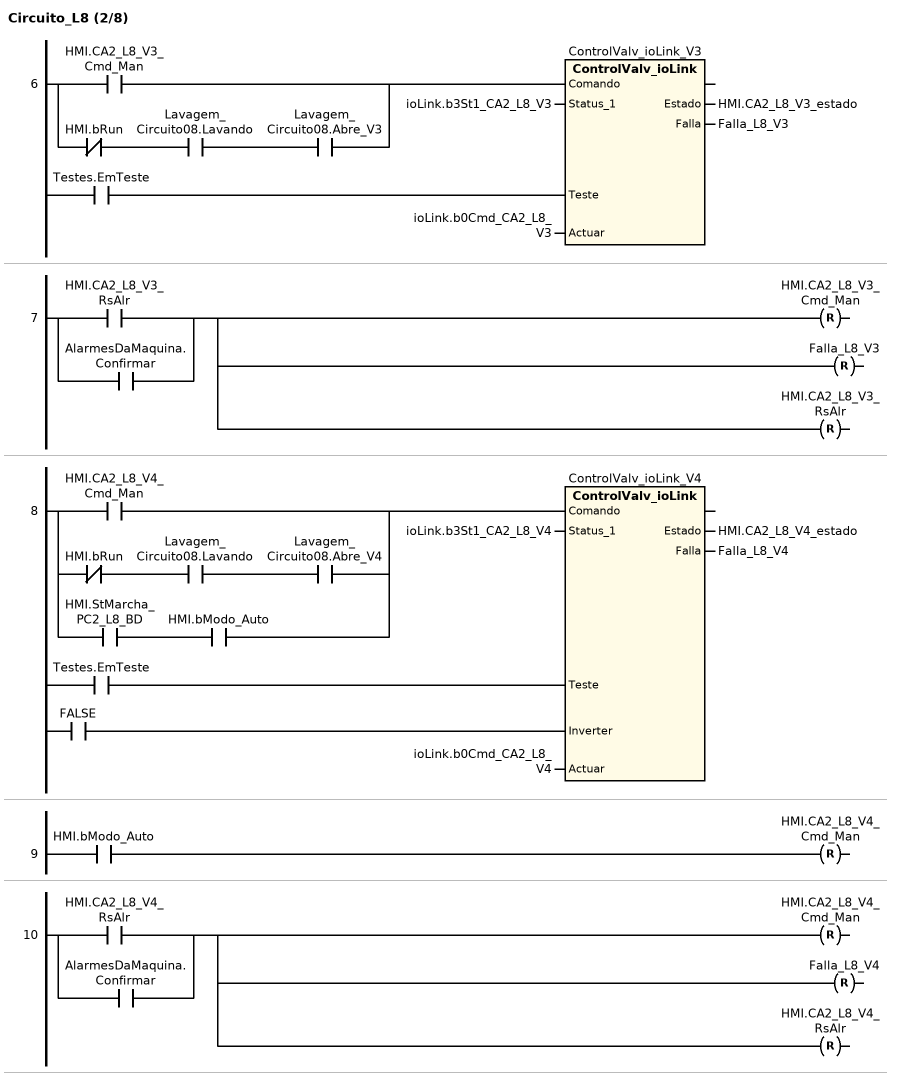
// NETWORK 6
ControlValv_ioLink_V3(
    Comando := HMI.CA2_L8_V3_Cmd_Man OR NOT HMI.bRun AND Lavagem_Circuito08.Lavando AND Lavagem_Circuito08.Abre_V3,
    Status_1 := ioLink.b3St1_CA2_L8_V3,
    Teste := Testes.EmTeste,
    Actuar := ioLink.b0Cmd_CA2_L8_V3,
    Estado => HMI.CA2_L8_V3_estado,
    Falla => Falla_L8_V3); // ControlValv_ioLink

// NETWORK 7
_w3 := HMI.CA2_L8_V3_RsAlr OR AlarmesDaMaquina.Confirmar;
HMI.CA2_L8_V3_Cmd_Man R= _w3;
Falla_L8_V3 R= _w3;
HMI.CA2_L8_V3_RsAlr R= _w3;

// NETWORK 8
ControlValv_ioLink_V4(
    Comando := HMI.CA2_L8_V4_Cmd_Man OR NOT HMI.bRun AND Lavagem_Circuito08.Lavando AND Lavagem_Circuito08.Abre_V4 OR HMI.StMarcha_PC2_L8_BD AND HMI.bModo_Auto,
    Status_1 := ioLink.b3St1_CA2_L8_V4,
    Teste := Testes.EmTeste,
    Inverter := FALSE,
    Actuar := ioLink.b0Cmd_CA2_L8_V4,
    Estado => HMI.CA2_L8_V4_estado,
    Falla => Falla_L8_V4); // ControlValv_ioLink

// NETWORK 9
HMI.CA2_L8_V4_Cmd_Man R= HMI.bModo_Auto;

// NETWORK 10
_w4 := HMI.CA2_L8_V4_RsAlr OR AlarmesDaMaquina.Confirmar;
HMI.CA2_L8_V4_Cmd_Man R= _w4;
Falla_L8_V4 R= _w4;
HMI.CA2_L8_V4_RsAlr R= _w4;

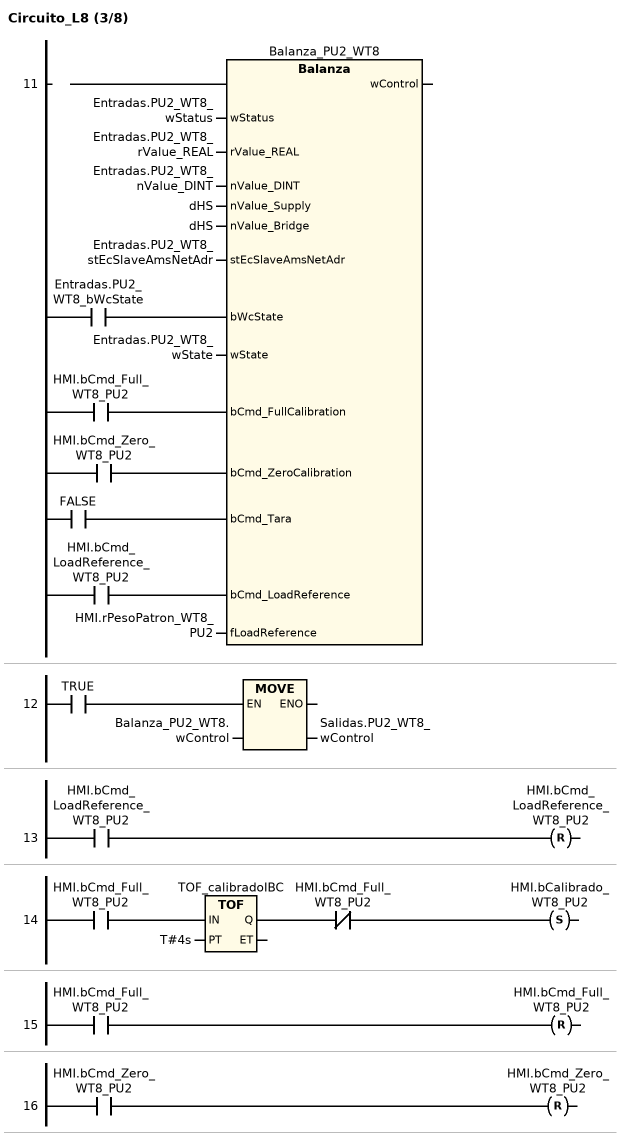
// NETWORK 11
Balanza_PU2_WT8(
    wStatus := Entradas.PU2_WT8_wStatus,
    rValue_REAL := Entradas.PU2_WT8_rValue_REAL,
    nValue_DINT := Entradas.PU2_WT8_nValue_DINT,
    nValue_Supply := dHS,
    nValue_Bridge := dHS,
    stEcSlaveAmsNetAdr := Entradas.PU2_WT8_stEcSlaveAmsNetAdr,
    bWcState := Entradas.PU2_WT8_bWcState,
    wState := Entradas.PU2_WT8_wState,
    bCmd_FullCalibration := HMI.bCmd_Full_WT8_PU2,
    bCmd_ZeroCalibration := HMI.bCmd_Zero_WT8_PU2,
    bCmd_Tara := FALSE,
    bCmd_LoadReference := HMI.bCmd_LoadReference_WT8_PU2,
    fLoadReference := HMI.rPesoPatron_WT8_PU2); // Balanza

// NETWORK 12
Salidas.PU2_WT8_wControl := Balanza_PU2_WT8.wControl;

// NETWORK 13
HMI.bCmd_LoadReference_WT8_PU2 R= HMI.bCmd_LoadReference_WT8_PU2;

// NETWORK 14
TOF_calibradoIBC(IN := HMI.bCmd_Full_WT8_PU2, PT := T#4s); // TOF
HMI.bCalibrado_WT8_PU2 S= TOF_calibradoIBC.Q AND NOT HMI.bCmd_Full_WT8_PU2;

// NETWORK 15
HMI.bCmd_Full_WT8_PU2 R= HMI.bCmd_Full_WT8_PU2;

// NETWORK 16
HMI.bCmd_Zero_WT8_PU2 R= HMI.bCmd_Zero_WT8_PU2;

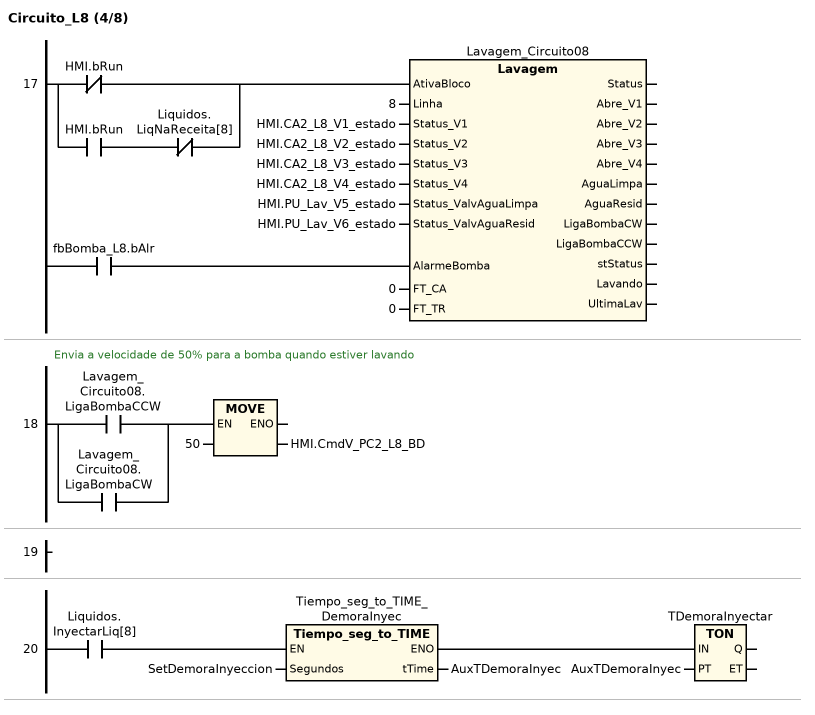
// NETWORK 17
Lavagem_Circuito08(
    AtivaBloco := NOT HMI.bRun OR HMI.bRun AND NOT Liquidos.LiqNaReceita[8],
    Linha := 8,
    Status_V1 := HMI.CA2_L8_V1_estado,
    Status_V2 := HMI.CA2_L8_V2_estado,
    Status_V3 := HMI.CA2_L8_V3_estado,
    Status_V4 := HMI.CA2_L8_V4_estado,
    Status_ValvAguaLimpa := HMI.PU_Lav_V5_estado,
    Status_ValvAguaResid := HMI.PU_Lav_V6_estado,
    AlarmeBomba := fbBomba_L8.bAlr,
    FT_CA := 0,
    FT_TR := 0); // Lavagem

// NETWORK 18
// Envia a velocidade de 50% para a bomba quando estiver lavando
IF Lavagem_Circuito08.LigaBombaCCW OR Lavagem_Circuito08.LigaBombaCW THEN HMI.CmdV_PC2_L8_BD := 50; END_IF

// NETWORK 19

// NETWORK 20
_w5 := Liquidos.InyectarLiq[8];
IF _w5 THEN
    Tiempo_seg_to_TIME_DemoraInyec(Segundos := SetDemoraInyeccion, tTime => AuxTDemoraInyec); // Tiempo_seg_to_TIME
END_IF
TDemoraInyectar(IN := _w5, PT := AuxTDemoraInyec); // TON

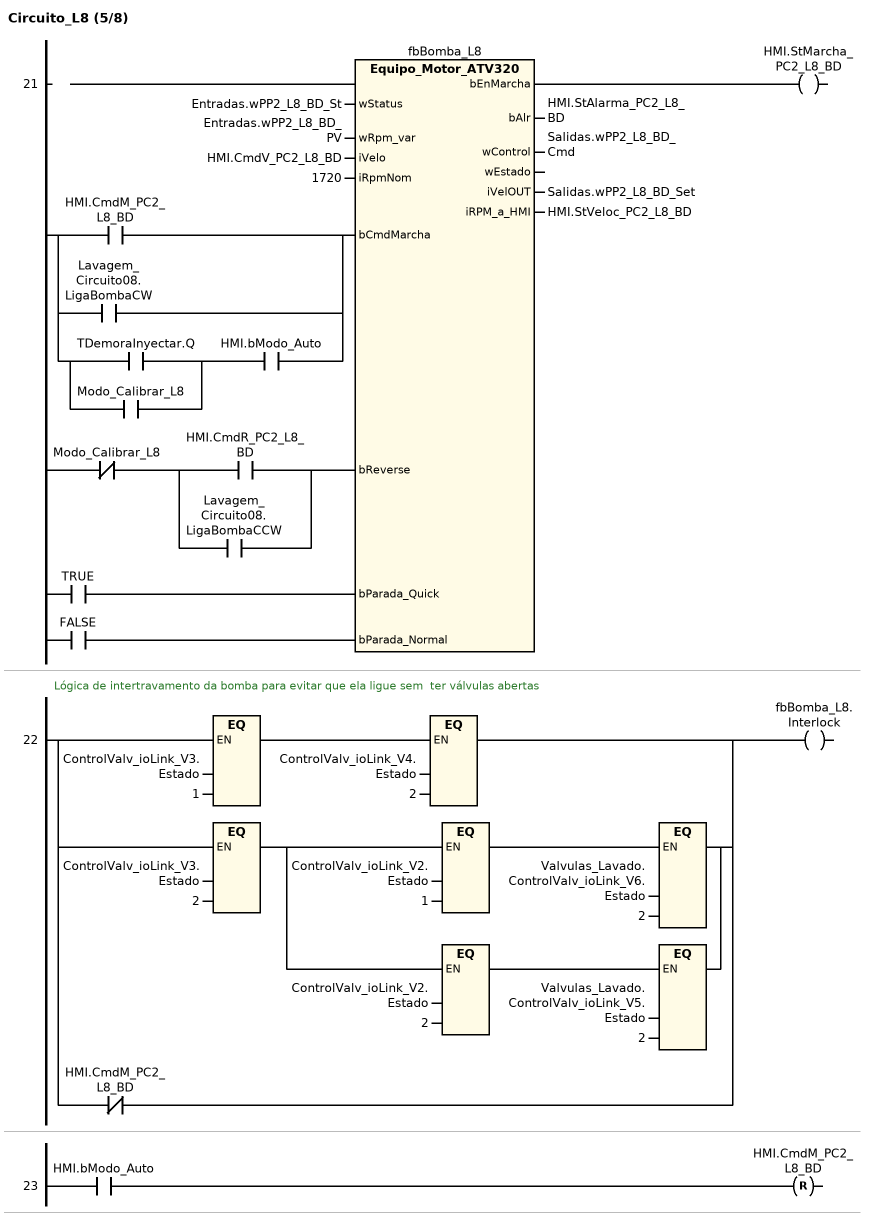
// NETWORK 21
fbBomba_L8(
    wStatus := Entradas.wPP2_L8_BD_St,
    wRpm_var := Entradas.wPP2_L8_BD_PV,
    iVelo := HMI.CmdV_PC2_L8_BD,
    iRpmNom := 1720,
    bCmdMarcha := HMI.CmdM_PC2_L8_BD OR Lavagem_Circuito08.LigaBombaCW OR (TDemoraInyectar.Q OR Modo_Calibrar_L8) AND HMI.bModo_Auto,
    bReverse := NOT Modo_Calibrar_L8 AND (HMI.CmdR_PC2_L8_BD OR Lavagem_Circuito08.LigaBombaCCW),
    bParada_Quick := TRUE,
    bParada_Normal := FALSE,
    bAlr => HMI.StAlarma_PC2_L8_BD,
    wControl => Salidas.wPP2_L8_BD_Cmd,
    iVelOUT => Salidas.wPP2_L8_BD_Set,
    iRPM_a_HMI => HMI.StVeloc_PC2_L8_BD); // Equipo_Motor_ATV320
HMI.StMarcha_PC2_L8_BD := fbBomba_L8.bEnMarcha;

// NETWORK 22
// Lógica de intertravamento da bomba para evitar que ela ligue sem  ter válvulas abertas
_w6 := NOT HMI.CmdM_PC2_L8_BD;
IF NOT _w6 THEN
    _w7 := ControlValv_ioLink_V3.Estado = 2;
    _w6 := ControlValv_ioLink_V3.Estado = 1 AND ControlValv_ioLink_V4.Estado = 2 OR (_w7 AND ControlValv_ioLink_V2.Estado = 1 AND Valvulas_Lavado.ControlValv_ioLink_V6.Estado = 2 OR _w7 AND ControlValv_ioLink_V2.Estado = 2 AND Valvulas_Lavado.ControlValv_ioLink_V5.Estado = 2);
END_IF
fbBomba_L8.Interlock := _w6;

// NETWORK 23
HMI.CmdM_PC2_L8_BD R= HMI.bModo_Auto;

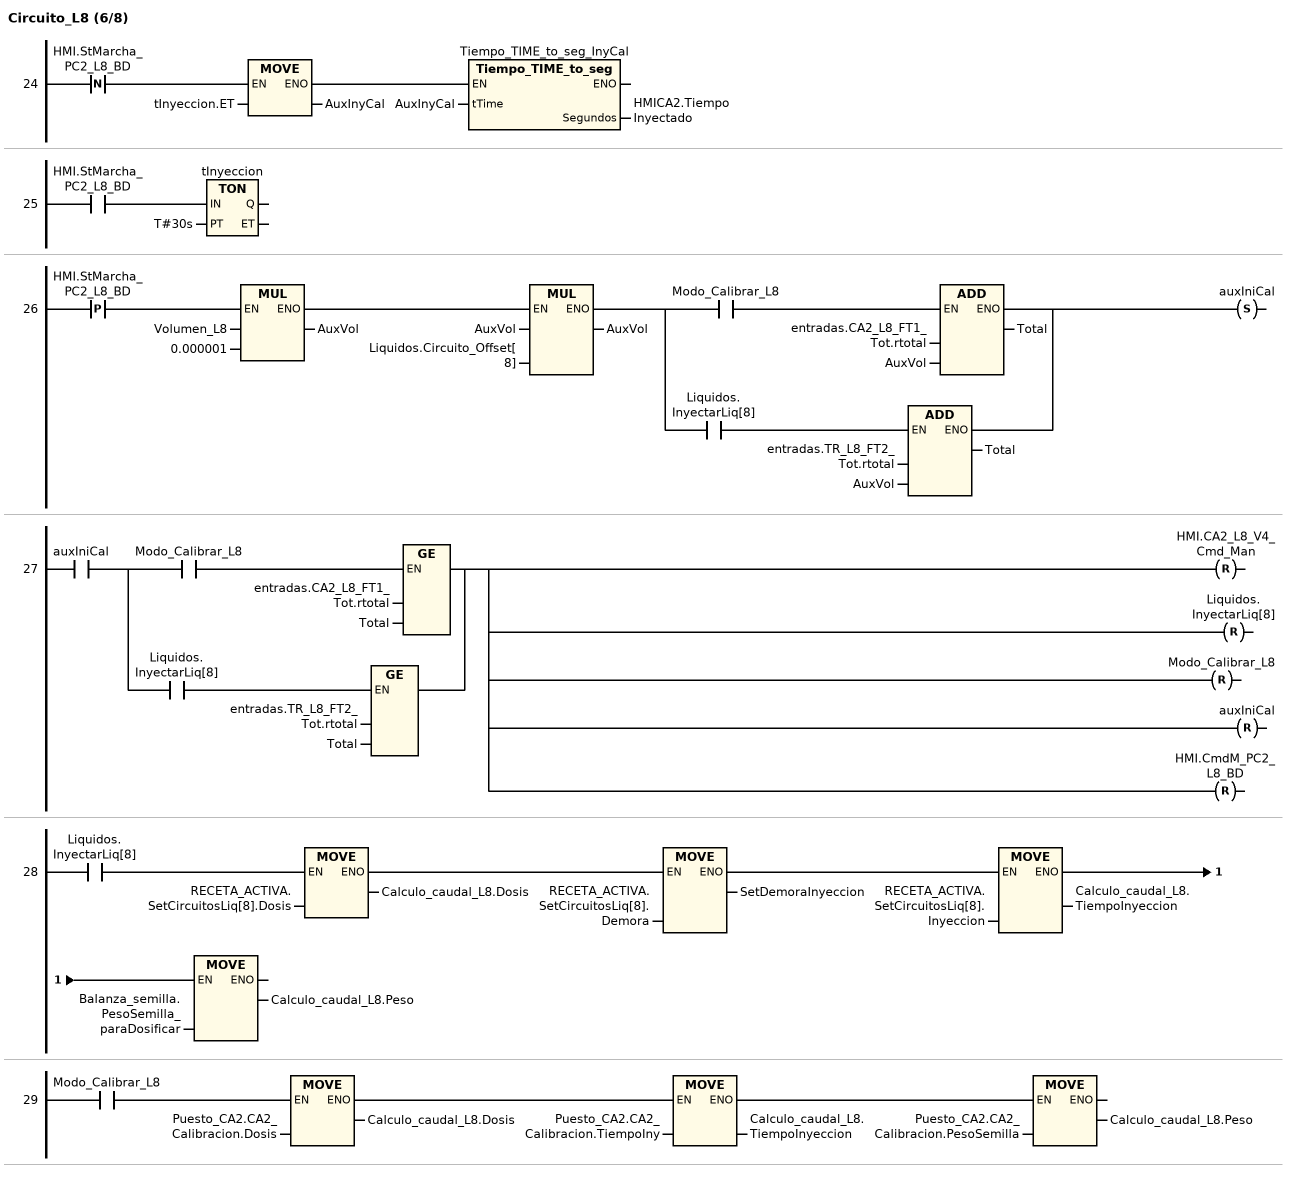
// NETWORK 24
_ft1(CLK := HMI.StMarcha_PC2_L8_BD);
_w8 := _ft1.Q;
IF _w8 THEN AuxInyCal := tInyeccion.ET; END_IF
IF _w8 THEN
    Tiempo_TIME_to_seg_InyCal(tTime := AuxInyCal, Segundos => HMICA2.TiempoInyectado); // Tiempo_TIME_to_seg
END_IF

// NETWORK 25
tInyeccion(IN := HMI.StMarcha_PC2_L8_BD, PT := T#30s); // TON

// NETWORK 26
_rt1(CLK := HMI.StMarcha_PC2_L8_BD);
_w9 := _rt1.Q;
IF _w9 THEN AuxVol := Volumen_L8 * 0.000001; END_IF
IF _w9 THEN AuxVol := AuxVol * Liquidos.Circuito_Offset[8]; END_IF
IF _w9 AND Modo_Calibrar_L8 THEN Total := entradas.CA2_L8_FT1_Tot.rtotal + AuxVol; END_IF
IF _w9 AND Liquidos.InyectarLiq[8] THEN Total := entradas.TR_L8_FT2_Tot.rtotal + AuxVol; END_IF
auxIniCal S= _w9 AND Modo_Calibrar_L8 OR _w9 AND Liquidos.InyectarLiq[8];

// NETWORK 27
_w10 := auxIniCal AND Modo_Calibrar_L8 AND entradas.CA2_L8_FT1_Tot.rtotal >= Total OR auxIniCal AND Liquidos.InyectarLiq[8] AND entradas.TR_L8_FT2_Tot.rtotal >= Total;
HMI.CA2_L8_V4_Cmd_Man R= _w10;
Liquidos.InyectarLiq[8] R= _w10;
Modo_Calibrar_L8 R= _w10;
auxIniCal R= _w10;
HMI.CmdM_PC2_L8_BD R= _w10;

// NETWORK 28
_w11 := Liquidos.InyectarLiq[8];
IF _w11 THEN Calculo_caudal_L8.Dosis := RECETA_ACTIVA.SetCircuitosLiq[8].Dosis; END_IF
IF _w11 THEN SetDemoraInyeccion := RECETA_ACTIVA.SetCircuitosLiq[8].Demora; END_IF
IF _w11 THEN Calculo_caudal_L8.TiempoInyeccion := RECETA_ACTIVA.SetCircuitosLiq[8].Inyeccion; END_IF
IF _w11 THEN Calculo_caudal_L8.Peso := Balanza_semilla.PesoSemilla_paraDosificar; END_IF

// NETWORK 29
_w12 := Modo_Calibrar_L8;
IF _w12 THEN Calculo_caudal_L8.Dosis := Puesto_CA2.CA2_Calibracion.Dosis; END_IF
IF _w12 THEN Calculo_caudal_L8.TiempoInyeccion := Puesto_CA2.CA2_Calibracion.TiempoIny; END_IF
IF _w12 THEN Calculo_caudal_L8.Peso := Puesto_CA2.CA2_Calibracion.PesoSemilla; END_IF

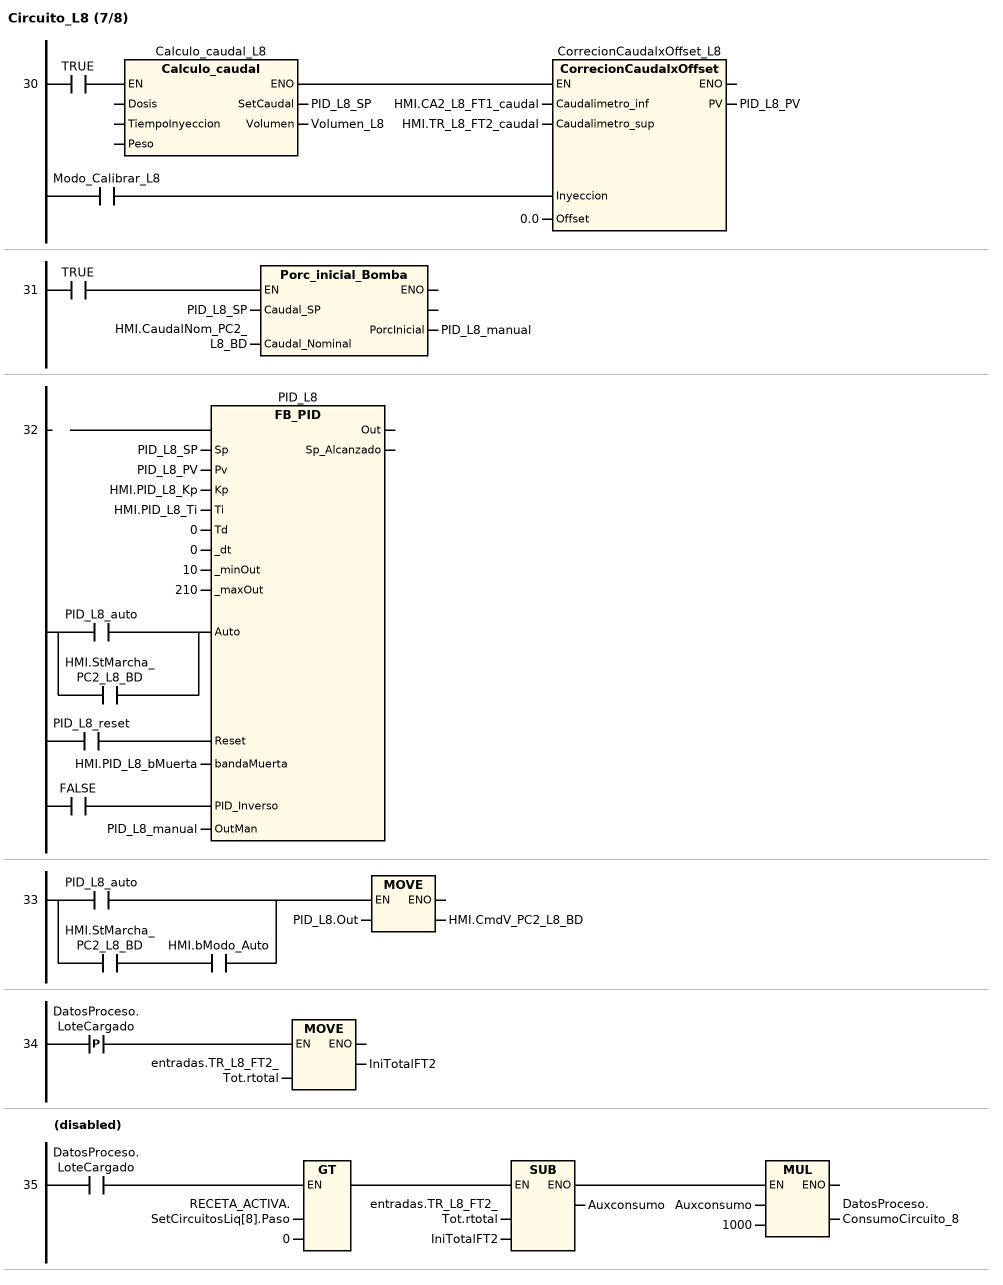
// NETWORK 30
Calculo_caudal_L8(SetCaudal => PID_L8_SP, Volumen => Volumen_L8); // Calculo_caudal
CorrecionCaudalxOffset_L8(
    Caudalimetro_inf := HMI.CA2_L8_FT1_caudal,
    Caudalimetro_sup := HMI.TR_L8_FT2_caudal,
    Inyeccion := Modo_Calibrar_L8,
    Offset := 0.0,
    PV => PID_L8_PV); // CorrecionCaudalxOffset

// NETWORK 31
Porc_inicial_Bomba(Caudal_SP := PID_L8_SP, Caudal_Nominal := HMI.CaudalNom_PC2_L8_BD, PorcInicial => PID_L8_manual);

// NETWORK 32
PID_L8(
    Sp := PID_L8_SP,
    Pv := PID_L8_PV,
    Kp := HMI.PID_L8_Kp,
    Ti := HMI.PID_L8_Ti,
    Td := 0,
    _dt := 0,
    _minOut := 10,
    _maxOut := 210,
    Auto := PID_L8_auto OR HMI.StMarcha_PC2_L8_BD,
    Reset := PID_L8_reset,
    bandaMuerta := HMI.PID_L8_bMuerta,
    PID_Inverso := FALSE,
    OutMan := PID_L8_manual); // FB_PID

// NETWORK 33
IF PID_L8_auto OR HMI.StMarcha_PC2_L8_BD AND HMI.bModo_Auto THEN HMI.CmdV_PC2_L8_BD := PID_L8.Out; END_IF

// NETWORK 34
_rt2(CLK := DatosProceso.LoteCargado);
IF _rt2.Q THEN IniTotalFT2 := entradas.TR_L8_FT2_Tot.rtotal; END_IF

// NETWORK 35 (disabled)
// _w13 := DatosProceso.LoteCargado AND RECETA_ACTIVA.SetCircuitosLiq[8].Paso > 0;
// IF _w13 THEN Auxconsumo := entradas.TR_L8_FT2_Tot.rtotal - IniTotalFT2; END_IF
// IF _w13 THEN DatosProceso.ConsumoCircuito_8 := Auxconsumo * 1000; END_IF

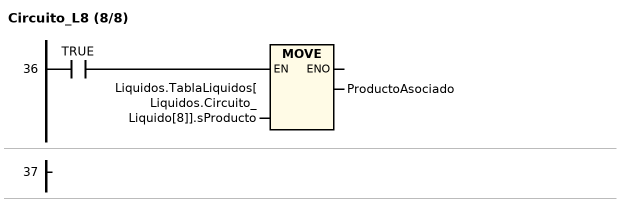
// NETWORK 36
ProductoAsociado := Liquidos.TablaLiquidos[Liquidos.Circuito_Liquido[8]].sProducto;

// NETWORK 37

END_PROGRAM

// ---- POUs/Puesto_Calibracion_3/Circuito_L9.TcPOU
PROGRAM Circuito_L9
VAR_INPUT
	Modo_Calibrar_L9: BOOL;
END_VAR
VAR
		fbBomba_L9 :Equipo_Motor_ATV320;
		ControlValv_ioLink_V1:ControlValv_ioLink;
		ControlValv_ioLink_V2: ControlValv_ioLink;
		ControlValv_ioLink_V3: ControlValv_ioLink;
		ControlValv_ioLink_V4: ControlValv_ioLink;
		Falla_L9_V1:BOOL;
		Falla_L9_V2:BOOL;
		Falla_L9_V3:BOOL;
		Falla_L9_V4:BOOL;
	Balanza_PU3_WT9: Balanza;
		dHS:DINT;
		TOF_calibradoIBC: TOF;
		AuxFinCalibrar:BOOL;
		PID_L9_SP:REAL;
		PID_L9_auto:BOOL;
		PID_L9_reset:BOOL;
		PID_L9_manual:REAL;
		PID_L9_bMuerta:REAL := 5;
		PID_L9_Kp:REAL := 0.1;
		PID_L9_Ti:REAL := 100;
		PID_L9_PV:REAL;
		Dosis_L9	:REAL;
		TiempoInyeccion_L9	:DINT;
		Peso	:REAL;
		Offset_L9:REAL;
		Inyeccion_L9:BOOL;

		Volumen_L9:REAL;
	Calculo_caudal_L9: Calculo_caudal;
	CorrecionCaudalxOffset_L9: CorrecionCaudalxOffset;
	tInyeccion: TON;
	Total :REAL;
	Totalant	:REAL;
	auxIniCal:BOOL;
	AuxVol9:REAL;
	TDemoraInyectar: TON;
	SetDemoraInyeccion: REAL;
	Tiempo_seg_to_TIME_DemoraInyec: Tiempo_seg_to_TIME;
	AuxTDemoraInyec: TIME;
	PID_L9: FB_PID;
	Tiempo_TIME_to_seg_InyCal: Tiempo_TIME_to_seg;
	AuxInyCal:TIME;
	ProductoAsociado: STRING;
	Lavagem_Circuito9: Lavagem;
END_VAR

VAR PERSISTENT
	UltimaCalibracao	:UDINT;	//Data e hora da ultima calibração
END_VAR
VAR // added by the converter: edge detectors and wires of the graphical bodies
    _w1, _w2, _w3, _w4, _w5, _w6, _w7, _w8, _w9, _w10, _w11, _w12 : BOOL;
    _ft1 : F_TRIG;
    _rt1 : R_TRIG;
END_VAR

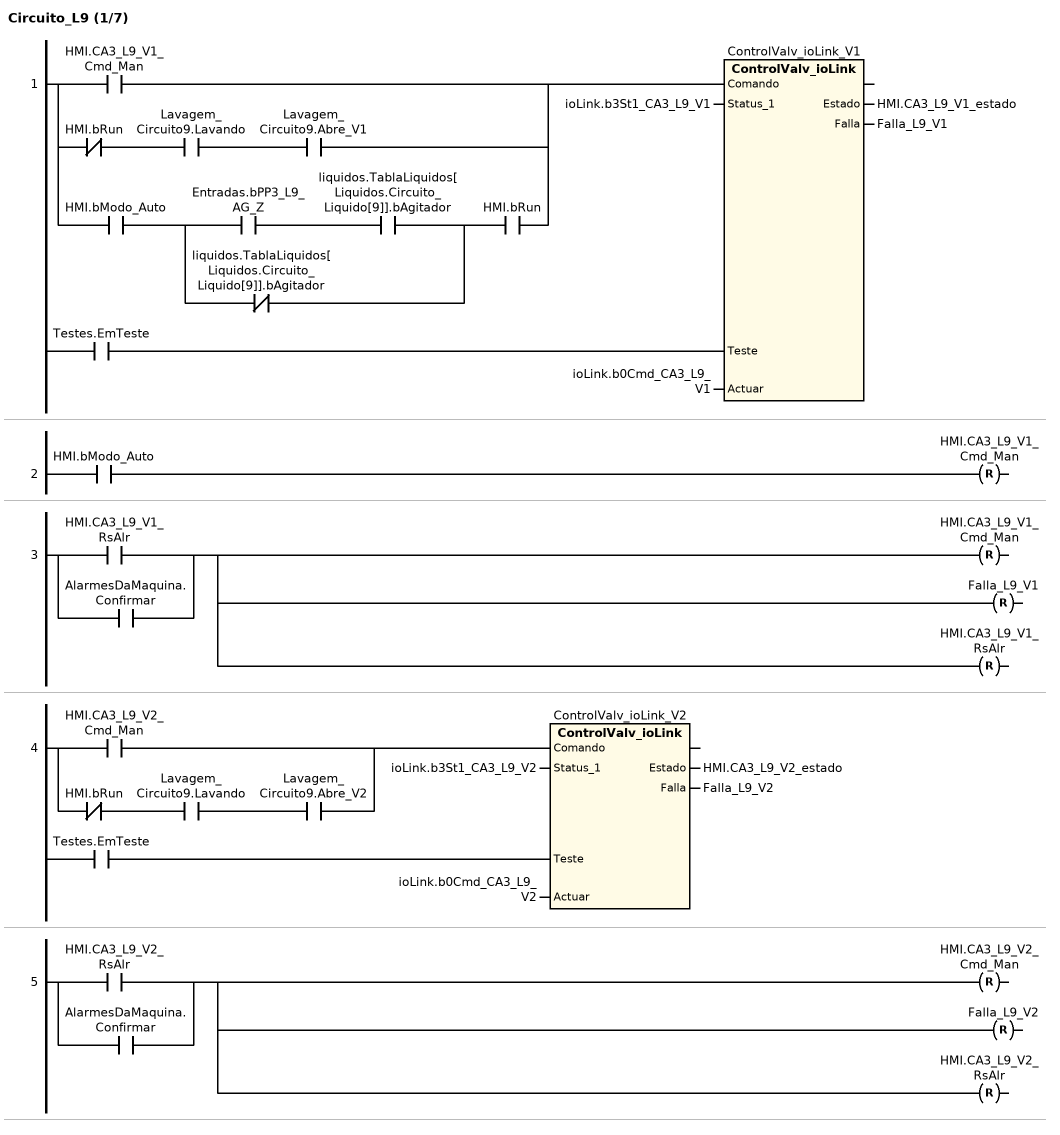
// NETWORK 1
ControlValv_ioLink_V1(
    Comando := HMI.CA3_L9_V1_Cmd_Man OR NOT HMI.bRun AND Lavagem_Circuito9.Lavando AND Lavagem_Circuito9.Abre_V1 OR HMI.bModo_Auto AND (Entradas.bPP3_L9_AG_Z AND (liquidos.TablaLiquidos[Liquidos.Circuito_Liquido[9]].bAgitador) OR NOT (liquidos.TablaLiquidos[Liquidos.Circuito_Liquido[9]].bAgitador)) AND HMI.bRun,
    Status_1 := ioLink.b3St1_CA3_L9_V1,
    Teste := Testes.EmTeste,
    Actuar := ioLink.b0Cmd_CA3_L9_V1,
    Estado => HMI.CA3_L9_V1_estado,
    Falla => Falla_L9_V1); // ControlValv_ioLink

// NETWORK 2
HMI.CA3_L9_V1_Cmd_Man R= HMI.bModo_Auto;

// NETWORK 3
_w1 := HMI.CA3_L9_V1_RsAlr OR AlarmesDaMaquina.Confirmar;
HMI.CA3_L9_V1_Cmd_Man R= _w1;
Falla_L9_V1 R= _w1;
HMI.CA3_L9_V1_RsAlr R= _w1;

// NETWORK 4
ControlValv_ioLink_V2(
    Comando := HMI.CA3_L9_V2_Cmd_Man OR NOT HMI.bRun AND Lavagem_Circuito9.Lavando AND Lavagem_Circuito9.Abre_V2,
    Status_1 := ioLink.b3St1_CA3_L9_V2,
    Teste := Testes.EmTeste,
    Actuar := ioLink.b0Cmd_CA3_L9_V2,
    Estado => HMI.CA3_L9_V2_estado,
    Falla => Falla_L9_V2); // ControlValv_ioLink

// NETWORK 5
_w2 := HMI.CA3_L9_V2_RsAlr OR AlarmesDaMaquina.Confirmar;
HMI.CA3_L9_V2_Cmd_Man R= _w2;
Falla_L9_V2 R= _w2;
HMI.CA3_L9_V2_RsAlr R= _w2;

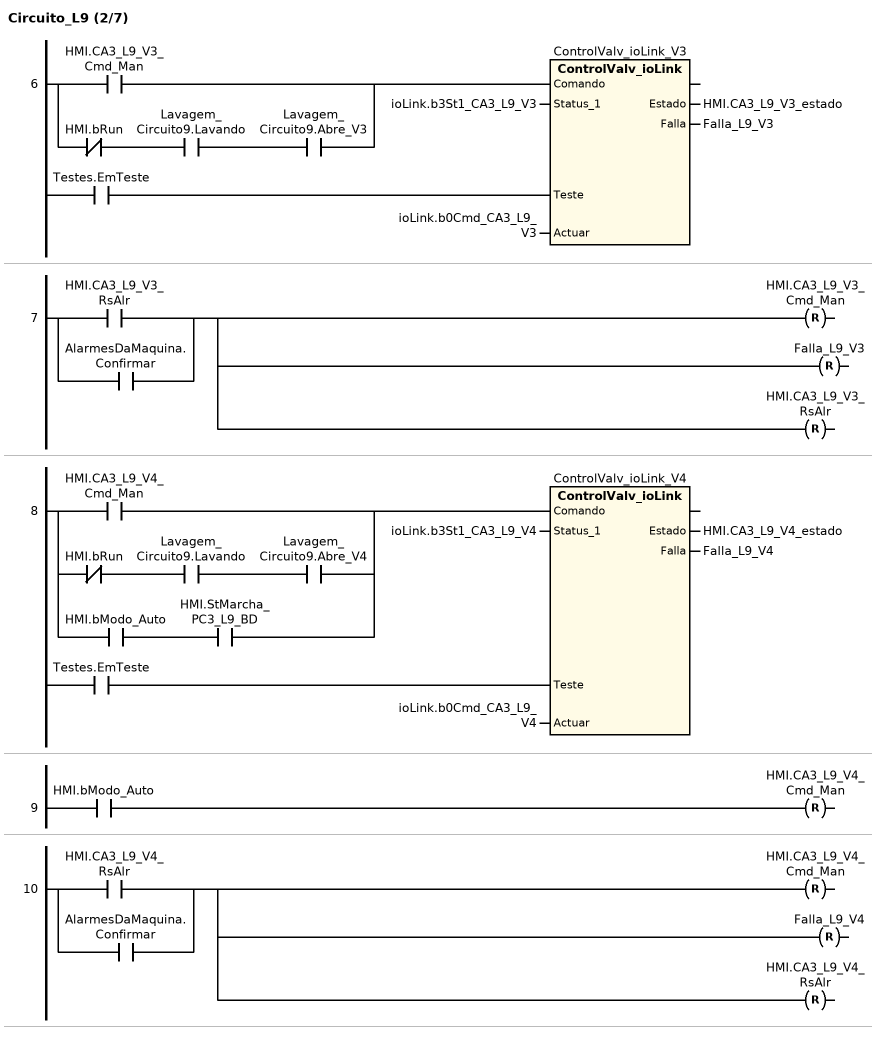
// NETWORK 6
ControlValv_ioLink_V3(
    Comando := HMI.CA3_L9_V3_Cmd_Man OR NOT HMI.bRun AND Lavagem_Circuito9.Lavando AND Lavagem_Circuito9.Abre_V3,
    Status_1 := ioLink.b3St1_CA3_L9_V3,
    Teste := Testes.EmTeste,
    Actuar := ioLink.b0Cmd_CA3_L9_V3,
    Estado => HMI.CA3_L9_V3_estado,
    Falla => Falla_L9_V3); // ControlValv_ioLink

// NETWORK 7
_w3 := HMI.CA3_L9_V3_RsAlr OR AlarmesDaMaquina.Confirmar;
HMI.CA3_L9_V3_Cmd_Man R= _w3;
Falla_L9_V3 R= _w3;
HMI.CA3_L9_V3_RsAlr R= _w3;

// NETWORK 8
ControlValv_ioLink_V4(
    Comando := HMI.CA3_L9_V4_Cmd_Man OR NOT HMI.bRun AND Lavagem_Circuito9.Lavando AND Lavagem_Circuito9.Abre_V4 OR HMI.bModo_Auto AND HMI.StMarcha_PC3_L9_BD,
    Status_1 := ioLink.b3St1_CA3_L9_V4,
    Teste := Testes.EmTeste,
    Actuar := ioLink.b0Cmd_CA3_L9_V4,
    Estado => HMI.CA3_L9_V4_estado,
    Falla => Falla_L9_V4); // ControlValv_ioLink

// NETWORK 9
HMI.CA3_L9_V4_Cmd_Man R= HMI.bModo_Auto;

// NETWORK 10
_w4 := HMI.CA3_L9_V4_RsAlr OR AlarmesDaMaquina.Confirmar;
HMI.CA3_L9_V4_Cmd_Man R= _w4;
Falla_L9_V4 R= _w4;
HMI.CA3_L9_V4_RsAlr R= _w4;

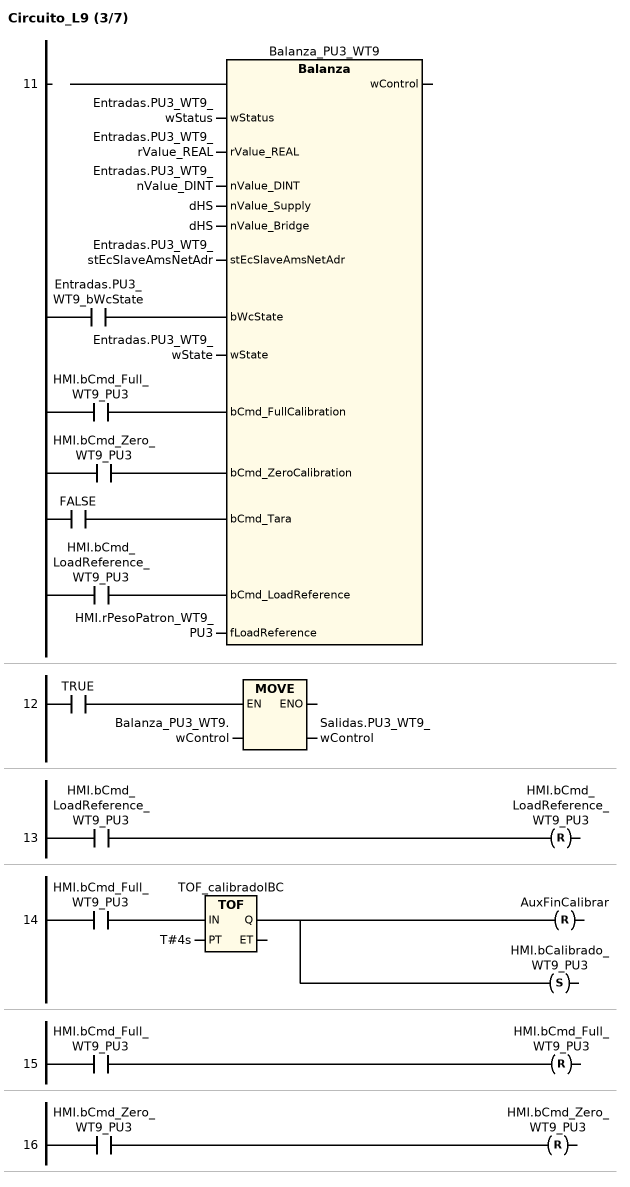
// NETWORK 11
Balanza_PU3_WT9(
    wStatus := Entradas.PU3_WT9_wStatus,
    rValue_REAL := Entradas.PU3_WT9_rValue_REAL,
    nValue_DINT := Entradas.PU3_WT9_nValue_DINT,
    nValue_Supply := dHS,
    nValue_Bridge := dHS,
    stEcSlaveAmsNetAdr := Entradas.PU3_WT9_stEcSlaveAmsNetAdr,
    bWcState := Entradas.PU3_WT9_bWcState,
    wState := Entradas.PU3_WT9_wState,
    bCmd_FullCalibration := HMI.bCmd_Full_WT9_PU3,
    bCmd_ZeroCalibration := HMI.bCmd_Zero_WT9_PU3,
    bCmd_Tara := FALSE,
    bCmd_LoadReference := HMI.bCmd_LoadReference_WT9_PU3,
    fLoadReference := HMI.rPesoPatron_WT9_PU3); // Balanza

// NETWORK 12
Salidas.PU3_WT9_wControl := Balanza_PU3_WT9.wControl;

// NETWORK 13
HMI.bCmd_LoadReference_WT9_PU3 R= HMI.bCmd_LoadReference_WT9_PU3;

// NETWORK 14
TOF_calibradoIBC(IN := HMI.bCmd_Full_WT9_PU3, PT := T#4s); // TOF
AuxFinCalibrar R= TOF_calibradoIBC.Q;
HMI.bCalibrado_WT9_PU3 S= TOF_calibradoIBC.Q;

// NETWORK 15
HMI.bCmd_Full_WT9_PU3 R= HMI.bCmd_Full_WT9_PU3;

// NETWORK 16
HMI.bCmd_Zero_WT9_PU3 R= HMI.bCmd_Zero_WT9_PU3;

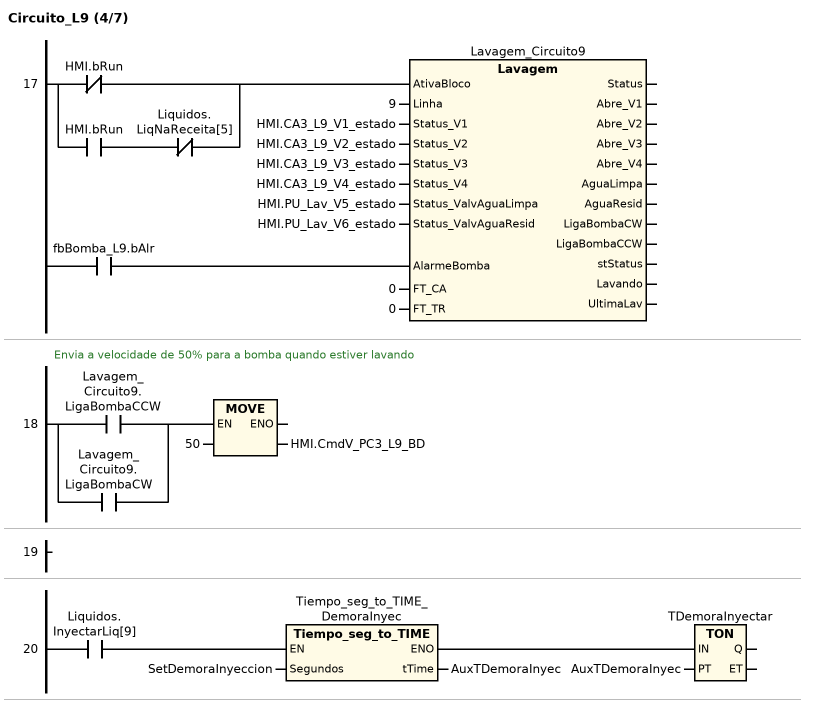
// NETWORK 17
Lavagem_Circuito9(
    AtivaBloco := NOT HMI.bRun OR HMI.bRun AND NOT Liquidos.LiqNaReceita[5],
    Linha := 9,
    Status_V1 := HMI.CA3_L9_V1_estado,
    Status_V2 := HMI.CA3_L9_V2_estado,
    Status_V3 := HMI.CA3_L9_V3_estado,
    Status_V4 := HMI.CA3_L9_V4_estado,
    Status_ValvAguaLimpa := HMI.PU_Lav_V5_estado,
    Status_ValvAguaResid := HMI.PU_Lav_V6_estado,
    AlarmeBomba := fbBomba_L9.bAlr,
    FT_CA := 0,
    FT_TR := 0); // Lavagem

// NETWORK 18
// Envia a velocidade de 50% para a bomba quando estiver lavando
IF Lavagem_Circuito9.LigaBombaCCW OR Lavagem_Circuito9.LigaBombaCW THEN HMI.CmdV_PC3_L9_BD := 50; END_IF

// NETWORK 19

// NETWORK 20
_w5 := Liquidos.InyectarLiq[9];
IF _w5 THEN
    Tiempo_seg_to_TIME_DemoraInyec(Segundos := SetDemoraInyeccion, tTime => AuxTDemoraInyec); // Tiempo_seg_to_TIME
END_IF
TDemoraInyectar(IN := _w5, PT := AuxTDemoraInyec); // TON

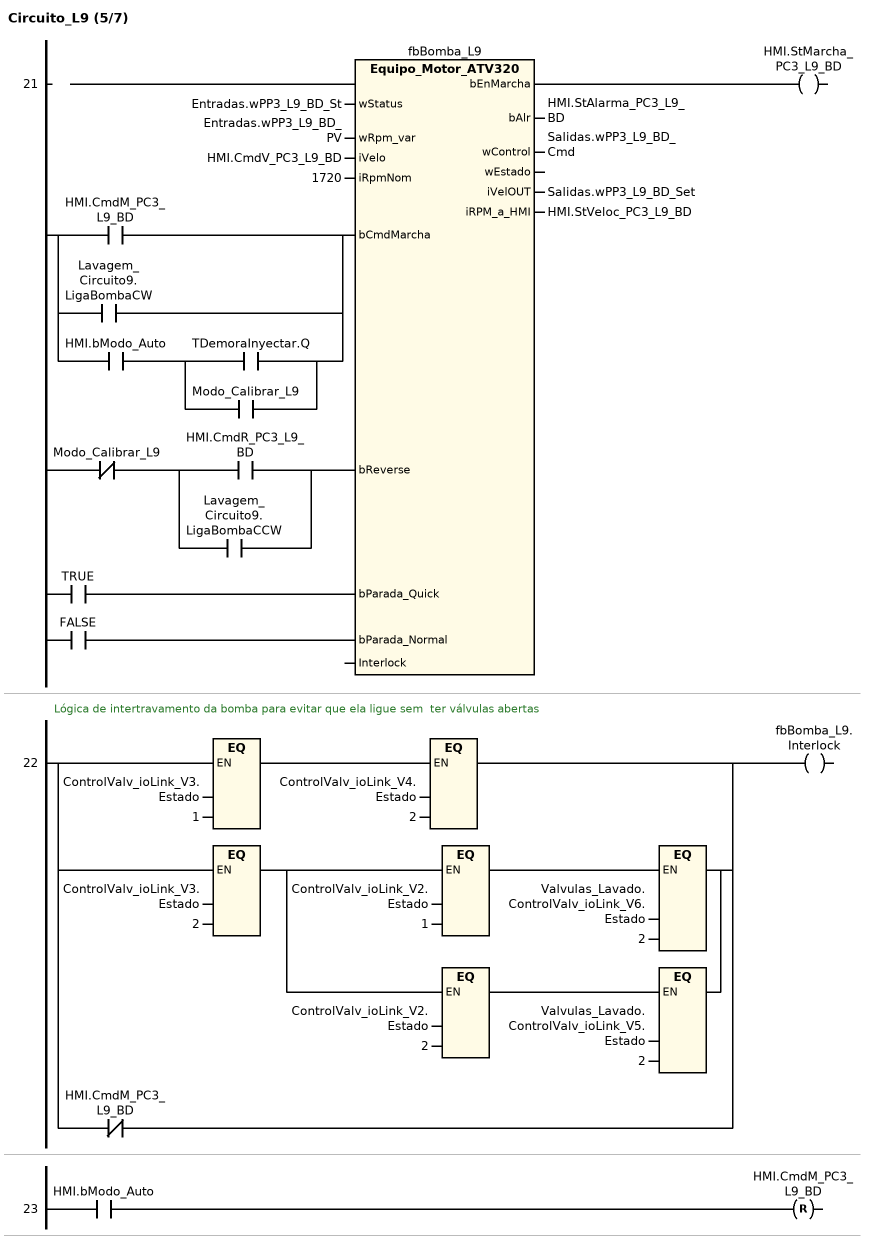
// NETWORK 21
fbBomba_L9(
    wStatus := Entradas.wPP3_L9_BD_St,
    wRpm_var := Entradas.wPP3_L9_BD_PV,
    iVelo := HMI.CmdV_PC3_L9_BD,
    iRpmNom := 1720,
    bCmdMarcha := HMI.CmdM_PC3_L9_BD OR Lavagem_Circuito9.LigaBombaCW OR HMI.bModo_Auto AND (TDemoraInyectar.Q OR Modo_Calibrar_L9),
    bReverse := NOT Modo_Calibrar_L9 AND (HMI.CmdR_PC3_L9_BD OR Lavagem_Circuito9.LigaBombaCCW),
    bParada_Quick := TRUE,
    bParada_Normal := FALSE,
    bAlr => HMI.StAlarma_PC3_L9_BD,
    wControl => Salidas.wPP3_L9_BD_Cmd,
    iVelOUT => Salidas.wPP3_L9_BD_Set,
    iRPM_a_HMI => HMI.StVeloc_PC3_L9_BD); // Equipo_Motor_ATV320
HMI.StMarcha_PC3_L9_BD := fbBomba_L9.bEnMarcha;

// NETWORK 22
// Lógica de intertravamento da bomba para evitar que ela ligue sem  ter válvulas abertas
_w6 := NOT HMI.CmdM_PC3_L9_BD;
IF NOT _w6 THEN
    _w7 := ControlValv_ioLink_V3.Estado = 2;
    _w6 := ControlValv_ioLink_V3.Estado = 1 AND ControlValv_ioLink_V4.Estado = 2 OR (_w7 AND ControlValv_ioLink_V2.Estado = 1 AND Valvulas_Lavado.ControlValv_ioLink_V6.Estado = 2 OR _w7 AND ControlValv_ioLink_V2.Estado = 2 AND Valvulas_Lavado.ControlValv_ioLink_V5.Estado = 2);
END_IF
fbBomba_L9.Interlock := _w6;

// NETWORK 23
HMI.CmdM_PC3_L9_BD R= HMI.bModo_Auto;

